C01812=1233.003,73.028,-45.498,-178.669,5.411,148.541
C01813=1233.007,72.779,-45.481,-178.672,5.410,148.542
C01814=1233.012,72.530,-45.463,-178.674,5.409,148.542
C01815=1233.017,72.280,-45.445,-178.677,5.409,148.543
C01816=1233.022,72.031,-45.427,-178.679,5.408,148.544
C01817=1233.027,71.782,-45.409,-178.682,5.408,148.544
C01818=1233.031,71.532,-45.393,-178.684,5.407,148.545
C01819=1233.036,71.283,-45.375,-178.687,5.406,148.545
C01820=1233.041,71.033,-45.358,-178.689,5.406,148.546
C01821=1233.047,70.785,-45.340,-178.692,5.405,148.547
C01822=1233.051,70.536,-45.323,-178.695,5.404,148.547
C01823=1233.056,70.286,-45.305,-178.697,5.404,148.548
C01824=1233.061,70.037,-45.287,-178.700,5.403,148.549
C01825=1233.066,69.787,-45.270,-178.702,5.402,148.549
C01826=1233.070,69.538,-45.253,-178.705,5.402,148.550
C01827=1233.076,69.289,-45.235,-178.707,5.401,148.550
C01828=1233.081,69.039,-45.217,-178.710,5.400,148.551
C01829=1233.085,68.790,-45.201,-178.712,5.400,148.552
C01830=1233.090,68.541,-45.183,-178.715,5.399,148.552
C01831=1233.095,68.291,-45.165,-178.718,5.399,148.553
C01832=1233.100,68.042,-45.147,-178.720,5.398,148.553
C01833=1233.105,67.792,-45.131,-178.722,5.397,148.554
C01834=1233.109,67.543,-45.113,-178.725,5.397,148.555
C01835=1233.115,67.293,-45.096,-178.728,5.396,148.555
C01836=1233.119,67.044,-45.078,-178.730,5.396,148.556
C01837=1233.124,66.795,-45.061,-178.732,5.396,148.557
C01838=1233.130,66.546,-45.043,-178.735,5.395,148.557
C01839=1233.134,66.297,-45.027,-178.737,5.394,148.558
C01840=1233.139,66.048,-45.009,-178.740,5.394,148.558
C01841=1233.143,65.798,-44.992,-178.742,5.393,148.559
C01842=1233.149,65.548,-44.975,-178.745,5.392,148.560
C01843=1233.154,65.299,-44.957,-178.748,5.392,148.560
C01844=1233.158,65.050,-44.940,-178.750,5.391,148.561
C01845=1233.163,64.800,-44.922,-178.752,5.390,148.562
C01846=1233.168,64.551,-44.905,-178.755,5.390,148.562
C01847=1233.173,64.302,-44.889,-178.758,5.389,148.563
C01848=1233.178,64.053,-44.871,-178.760,5.388,148.564
C01849=1233.183,63.803,-44.854,-178.763,5.388,148.564
C01850=1233.188,63.553,-44.837,-178.766,5.387,148.565
C01851=1233.193,63.304,-44.819,-178.768,5.387,148.566
C01852=1233.197,63.055,-44.802,-178.770,5.386,148.566
C01853=1233.203,62.805,-44.785,-178.773,5.385,148.567
C01854=1233.207,62.557,-44.768,-178.776,5.385,148.567
C01855=1233.213,62.307,-44.750,-178.778,5.384,148.568
C01856=1233.217,62.058,-44.734,-178.781,5.383,148.569
C01857=1233.222,61.808,-44.716,-178.784,5.383,148.569
C01858=1233.227,61.559,-44.699,-178.786,5.382,148.570
C01859=1233.232,61.309,-44.682,-178.788,5.382,148.571
C01860=1233.237,61.060,-44.665,-178.790,5.382,148.571
C01861=1233.242,60.811,-44.648,-178.793,5.381,148.572
C01862=1233.247,60.561,-44.630,-178.796,5.380,148.572
C01863=1233.251,60.312,-44.614,-178.798,5.380,148.573
C01864=1233.257,60.062,-44.596,-178.801,5.379,148.574
C01865=1233.262,59.813,-44.580,-178.804,5.379,148.574
C01866=1233.267,59.564,-44.562,-178.806,5.378,148.575
C01867=1233.271,59.315,-44.545,-178.809,5.377,148.576
C01868=1233.276,59.065,-44.528,-178.811,5.377,148.576
C01869=1233.281,58.815,-44.511,-178.814,5.376,148.577
C01870=1233.287,58.566,-44.495,-178.816,5.375,148.578
C01871=1233.291,58.317,-44.477,-178.819,5.375,148.578
C01872=1233.296,58.068,-44.460,-178.821,5.374,148.579
C01873=1233.300,57.818,-44.443,-178.824,5.374,148.580
C01874=1233.305,57.569,-44.427,-178.826,5.374,148.580
C01875=1233.311,57.319,-44.410,-178.829,5.373,148.581
C01876=1233.315,57.070,-44.393,-178.831,5.373,148.582
C01877=1233.320,56.820,-44.376,-178.834,5.372,148.582
C01878=1233.325,56.571,-44.359,-178.836,5.371,148.583
C01879=1233.330,56.322,-44.341,-178.839,5.371,148.583
C01880=1233.335,56.053,-44.324,-178.842,5.370,148.584
C01881=1233.341,55.785,-44.306,-178.844,5.369,148.585
C01882=1233.346,55.516,-44.288,-178.847,5.369,148.586
C01883=1233.351,55.248,-44.270,-178.850,5.369,148.586
C01884=1233.356,54.999,-44.253,-178.853,5.368,148.587
C01885=1233.361,54.749,-44.236,-178.855,5.367,148.587
C01886=1233.366,54.499,-44.219,-178.857,5.367,148.588
C01887=1233.371,54.251,-44.202,-178.860,5.366,148.589
C01888=1233.376,54.001,-44.186,-178.863,5.365,148.589
C01889=1233.381,53.751,-44.168,-178.865,5.365,148.590
C01890=1233.385,53.502,-44.152,-178.868,5.364,148.591
C01891=1233.390,53.253,-44.136,-178.870,5.364,148.591
C01892=1233.396,53.003,-44.118,-178.873,5.364,148.592
C01893=1233.400,52.754,-44.102,-178.875,5.363,148.593
C01894=1233.405,52.505,-44.085,-178.878,5.363,148.593
C01895=1233.410,52.255,-44.068,-178.880,5.362,148.594
C01896=1233.415,52.006,-44.051,-178.883,5.361,148.594
C01897=1233.420,51.757,-44.035,-178.885,5.361,148.595
C01898=1233.425,51.507,-44.018,-178.888,5.360,148.596
C01899=1233.430,51.258,-44.001,-178.891,5.359,148.596
C01900=1233.435,51.009,-43.985,-178.893,5.359,148.597
C01901=1233.440,50.759,-43.968,-178.896,5.358,148.598
C01902=1233.445,50.510,-43.951,-178.898,5.359,148.598
C01903=1233.450,50.261,-43.935,-178.900,5.358,148.599
C01904=1233.454,50.011,-43.918,-178.903,5.357,148.600
C01905=1233.459,49.762,-43.901,-178.905,5.357,148.600
C01906=1233.465,49.512,-43.885,-178.908,5.356,148.601
C01907=1233.469,49.263,-43.868,-178.911,5.355,148.602
C01908=1233.474,49.013,-43.852,-178.913,5.355,148.602
C01909=1233.479,48.764,-43.835,-178.916,5.354,148.603
C01910=1233.484,48.515,-43.818,-178.918,5.354,148.604
C01911=1233.488,48.265,-43.801,-178.921,5.354,148.604
C01912=1233.493,48.016,-43.785,-178.923,5.353,148.605
C01913=1233.499,47.766,-43.769,-178.926,5.353,148.606
C01914=1233.504,47.517,-43.752,-178.928,5.352,148.606
C01915=1233.509,47.268,-43.736,-178.931,5.352,148.607
C01916=1233.513,47.018,-43.719,-178.934,5.351,148.608
C01917=1233.518,46.769,-43.703,-178.936,5.350,148.608
C01918=1233.524,46.519,-43.686,-178.938,5.350,148.609
C01919=1233.528,46.269,-43.669,-178.941,5.350,148.609
C01920=1233.533,46.021,-43.653,-178.943,5.349,148.610
C01921=1233.538,45.771,-43.636,-178.946,5.349,148.611
C01922=1233.543,45.522,-43.621,-178.948,5.348,148.611
C01923=1233.548,45.272,-43.604,-178.951,5.347,148.612
C01924=1233.553,45.023,-43.587,-178.954,5.347,148.613
C01925=1233.558,44.773,-43.571,-178.956,5.346,148.613
C01926=1233.563,44.524,-43.555,-178.959,5.346,148.614
C01927=1233.568,44.275,-43.538,-178.961,5.346,148.615
C01928=1233.572,44.025,-43.522,-178.964,5.345,148.615
C01929=1233.578,43.776,-43.506,-178.966,5.345,148.616
C01930=1233.583,43.526,-43.489,-178.969,5.344,148.617
C01931=1233.588,43.277,-43.473,-178.971,5.343,148.617
C01932=1233.593,43.027,-43.457,-178.974,5.343,148.618
C01933=1233.597,42.778,-43.440,-178.976,5.342,148.619
C01934=1233.602,42.529,-43.424,-178.979,5.342,148.619
C01935=1233.607,42.279,-43.408,-178.981,5.342,148.620
C01936=1233.612,42.030,-43.391,-178.984,5.341,148.621
C01937=1233.617,41.780,-43.375,-178.986,5.341,148.621
C01938=1233.622,41.531,-43.359,-178.989,5.340,148.622
C01939=1233.626,41.282,-43.342,-178.992,5.340,148.623
C01940=1233.633,41.032,-43.326,-178.994,5.339,148.623
C01941=1233.637,40.783,-43.310,-178.996,5.339,148.624
C01942=1233.642,40.533,-43.294,-178.999,5.339,148.625
C01943=1233.647,40.284,-43.277,-179.002,5.338,148.625
C01944=1233.652,40.035,-43.261,-179.004,5.338,148.626
C01945=1233.657,39.785,-43.245,-179.007,5.337,148.627
C01946=1233.662,39.536,-43.229,-179.010,5.337,148.627
C01947=1233.667,39.286,-43.213,-179.012,5.336,148.628
C01948=1233.672,39.037,-43.197,-179.014,5.336,148.628
C01949=1233.677,38.787,-43.181,-179.016,5.335,148.629
C01950=1233.682,38.538,-43.164,-179.019,5.335,148.630
C01951=1233.686,38.288,-43.148,-179.022,5.334,148.631
C01952=1233.691,38.039,-43.132,-179.024,5.334,148.631
C01953=1233.696,37.789,-43.116,-179.027,5.333,148.632
C01954=1233.701,37.540,-43.100,-179.029,5.333,148.633
C01955=1233.706,37.290,-43.084,-179.032,5.333,148.633
C01956=1233.711,37.042,-43.068,-179.034,5.332,148.634
C01957=1233.716,36.791,-43.052,-179.037,5.332,148.635
C01958=1233.721,36.543,-43.035,-179.040,5.331,148.635
C01959=1233.726,36.293,-43.020,-179.042,5.330,148.636
C01960=1233.731,36.043,-43.004,-179.044,5.331,148.637
C01961=1233.736,35.794,-42.987,-179.047,5.330,148.637
C01962=1233.741,35.544,-42.971,-179.050,5.330,148.638
C01963=1233.746,35.296,-42.955,-179.052,5.329,148.639
C01964=1233.751,35.045,-42.939,-179.055,5.328,148.639
C01965=1233.756,34.796,-42.924,-179.058,5.328,148.640
C01966=1233.760,34.547,-42.908,-179.060,5.328,148.641
C01967=1233.766,34.297,-42.892,-179.062,5.328,148.641
C01968=1233.771,34.049,-42.876,-179.065,5.327,148.642
C01969=1233.775,33.799,-42.860,-179.067,5.326,148.642
C01970=1233.781,33.549,-42.844,-179.070,5.326,148.643
C01971=1233.785,33.300,-42.827,-179.072,5.325,148.644
C01972=1233.791,33.050,-42.812,-179.074,5.325,148.644
C01973=1233.796,32.801,-42.796,-179.077,5.325,148.645
C01974=1233.800,32.551,-42.780,-179.080,5.324,148.646
C01975=1233.805,32.302,-42.765,-179.082,5.324,148.647
C01976=1233.810,32.052,-42.749,-179.085,5.323,148.647
C01977=1233.815,31.803,-42.732,-179.087,5.323,148.648
C01978=1233.820,31.554,-42.717,-179.090,5.323,148.649
C01979=1233.825,31.304,-42.701,-179.092,5.322,148.649
C01980=1233.831,31.054,-42.685,-179.095,5.322,148.650
C01981=1233.835,30.805,-42.669,-179.098,5.321,148.651
C01982=1233.840,30.556,-42.654,-179.100,5.320,148.651
C01983=1233.845,30.307,-42.638,-179.102,5.321,148.652
C01984=1233.850,30.037,-42.621,-179.105,5.320,148.653
C01985=1233.856,29.769,-42.604,-179.108,5.320,148.653
C01986=1233.861,29.500,-42.587,-179.111,5.319,148.654
C01987=1233.867,29.232,-42.570,-179.113,5.319,148.655
C01988=1233.871,28.983,-42.555,-179.116,5.318,148.656
C01989=1233.876,28.733,-42.539,-179.119,5.318,148.656
C01990=1233.881,28.484,-42.522,-179.121,5.317,148.657
C01991=1233.887,28.235,-42.507,-179.123,5.317,148.658
C01992=1233.891,27.984,-42.491,-179.126,5.317,148.658
C01993=1233.896,27.735,-42.476,-179.129,5.316,148.659
C01994=1233.901,27.486,-42.460,-179.131,5.316,148.660
C01995=1233.906,27.236,-42.444,-179.134,5.315,148.660
C01996=1233.911,26.987,-42.428,-179.136,5.315,148.661
C01997=1233.916,26.738,-42.413,-179.139,5.315,148.662
C01998=1233.921,26.488,-42.397,-179.141,5.314,148.662
C01999=1233.926,26.238,-42.381,-179.144,5.314,148.663
C02000=1233.932,25.989,-42.366,-179.146,5.314,148.664
C02001=1233.936,25.739,-42.350,-179.148,5.313,148.664
C02002=1233.941,25.490,-42.335,-179.151,5.313,148.665
C02003=1233.946,25.240,-42.319,-179.154,5.312,148.666
C02004=1233.951,24.991,-42.304,-179.156,5.312,148.666
C02005=1233.955,24.742,-42.288,-179.158,5.312,148.667
C02006=1233.961,24.492,-42.272,-179.161,5.311,148.668
C02007=1233.966,24.243,-42.256,-179.164,5.311,148.668
C02008=1233.970,23.993,-42.241,-179.166,5.310,148.669
C02009=1233.976,23.744,-42.225,-179.169,5.310,148.670
C02010=1233.981,23.494,-42.210,-179.171,5.310,148.670
C02011=1233.986,23.245,-42.195,-179.174,5.309,148.671
C02012=1233.990,22.995,-42.179,-179.176,5.309,148.672
C02013=1233.996,22.746,-42.163,-179.179,5.308,148.672
C02014=1234.001,22.497,-42.148,-179.181,5.308,148.673
C02015=1234.006,22.247,-42.133,-179.184,5.308,148.674
C02016=1234.010,21.998,-42.117,-179.186,5.307,148.674
C02017=1234.015,21.748,-42.102,-179.189,5.307,148.675
C02018=1234.021,21.499,-42.086,-179.192,5.306,148.676
C02019=1234.025,21.250,-42.071,-179.194,5.306,148.676
C02020=1234.030,21.000,-42.055,-179.196,5.306,148.677
C02021=1234.036,20.750,-42.040,-179.199,5.305,148.678
C02022=1234.040,20.501,-42.025,-179.202,5.305,148.678
C02023=1234.046,20.251,-42.010,-179.204,5.305,148.679
C02024=1234.050,20.001,-41.994,-179.206,5.305,148.680
C02025=1234.055,19.752,-41.979,-179.209,5.304,148.681
C02026=1234.061,19.502,-41.963,-179.212,5.303,148.681
C02027=1234.065,19.253,-41.948,-179.214,5.303,148.682
C02028=1234.071,19.004,-41.933,-179.216,5.303,148.683
C02029=1234.075,18.754,-41.917,-179.219,5.303,148.683
C02030=1234.080,18.505,-41.902,-179.222,5.302,148.684
C02031=1234.085,18.256,-41.887,-179.224,5.302,148.685
C02032=1234.091,18.006,-41.872,-179.226,5.302,148.685
C02033=1234.095,17.757,-41.857,-179.229,5.301,148.686
C02034=1234.101,17.507,-41.841,-179.232,5.301,148.687
C02035=1234.105,17.257,-41.825,-179.234,5.300,148.687
C02036=1234.110,17.008,-41.810,-179.236,5.300,148.688
C02037=1234.115,16.759,-41.795,-179.239,5.300,148.689
C02038=1234.120,16.509,-41.781,-179.242,5.299,148.689
C02039=1234.126,16.259,-41.765,-179.244,5.299,148.690
C02040=1234.130,16.010,-41.750,-179.246,5.299,148.691
C02041=1234.135,15.760,-41.734,-179.249,5.299,148.691
C02042=1234.140,15.511,-41.719,-179.252,5.298,148.692
C02043=1234.146,15.261,-41.704,-179.254,5.297,148.693
C02044=1234.150,15.012,-41.689,-179.256,5.298,148.694
C02045=1234.156,14.763,-41.674,-179.259,5.297,148.694
C02046=1234.160,14.514,-41.659,-179.262,5.297,148.695
C02047=1234.166,14.264,-41.644,-179.264,5.296,148.696
C02048=1234.170,14.014,-41.628,-179.266,5.296,148.696
C02049=1234.175,13.765,-41.613,-179.269,5.296,148.697
C02050=1234.180,13.515,-41.598,-179.272,5.295,148.698
C02051=1234.185,13.266,-41.583,-179.274,5.295,148.698
C02052=1234.190,13.016,-41.568,-179.276,5.295,148.699
C02053=1234.195,12.767,-41.553,-179.279,5.294,148.700
C02054=1234.201,12.517,-41.538,-179.282,5.294,148.700
C02055=1234.205,12.268,-41.523,-179.284,5.293,148.701
C02056=1234.210,12.018,-41.507,-179.286,5.294,148.702
C02057=1234.215,11.768,-41.493,-179.289,5.293,148.702
C02058=1234.220,11.519,-41.478,-179.292,5.293,148.703
C02059=1234.225,11.270,-41.462,-179.294,5.292,148.704
C02060=1234.230,11.020,-41.448,-179.296,5.292,148.704
C02061=1234.235,10.771,-41.432,-179.300,5.292,148.705
C02062=1234.240,10.521,-41.417,-179.302,5.292,148.706
C02063=1234.245,10.272,-41.403,-179.305,5.291,148.707
C02064=1234.250,10.022,-41.387,-179.307,5.291,148.707
C02065=1234.255,9.773,-41.373,-179.310,5.291,148.708
C02066=1234.260,9.524,-41.358,-179.312,5.290,148.709
C02067=1234.265,9.274,-41.343,-179.314,5.290,148.710
C02068=1234.270,9.024,-41.328,-179.317,5.290,148.710
C02069=1234.274,8.775,-41.313,-179.320,5.289,148.711
C02070=1234.280,8.525,-41.298,-179.322,5.289,148.712
C02071=1234.285,8.275,-41.283,-179.324,5.289,148.712
C02072=1234.290,8.026,-41.269,-179.327,5.289,148.713
C02073=1234.295,7.776,-41.253,-179.330,5.288,148.714
C02074=1234.300,7.527,-41.239,-179.332,5.288,148.714
C02075=1234.305,7.278,-41.224,-179.334,5.288,148.715
C02076=1234.310,7.028,-41.209,-179.337,5.287,148.716
C02077=1234.315,6.778,-41.194,-179.340,5.287,148.716
C02078=1234.320,6.529,-41.180,-179.342,5.287,148.717
C02079=1234.325,6.279,-41.164,-179.344,5.286,148.718
C02080=1234.330,6.030,-41.150,-179.347,5.286,148.718
C02081=1234.335,5.781,-41.135,-179.350,5.285,148.719
C02082=1234.340,5.531,-41.121,-179.352,5.286,148.720
C02083=1234.345,5.281,-41.105,-179.354,5.285,148.720
C02084=1234.350,5.032,-41.091,-179.357,5.285,148.721
C02085=1234.355,4.783,-41.076,-179.359,5.285,148.722
C02086=1234.360,4.533,-41.062,-179.362,5.284,148.723
C02087=1234.365,4.284,-41.046,-179.364,5.284,148.723
C02088=1234.370,4.015,-41.030,-179.367,5.283,148.724
C02089=1234.376,3.746,-41.015,-179.370,5.283,148.725
C02090=1234.381,3.477,-40.998,-179.372,5.283,148.726
C02091=1234.387,3.207,-40.983,-179.375,5.283,148.726
C02092=1234.391,2.958,-40.968,-179.378,5.282,148.727
C02093=1234.396,2.709,-40.954,-179.380,5.282,148.728
C02094=1234.402,2.459,-40.938,-179.382,5.282,148.728
C02095=1234.407,2.210,-40.924,-179.385,5.282,148.729
C02096=1234.412,1.961,-40.910,-179.388,5.281,148.730
C02097=1234.417,1.711,-40.895,-179.390,5.281,148.730
C02098=1234.422,1.462,-40.881,-179.392,5.281,148.731
C02099=1234.428,1.212,-40.866,-179.395,5.280,148.732
C02100=1234.432,0.963,-40.851,-179.398,5.280,148.732
C02101=1234.437,0.713,-40.837,-179.400,5.280,148.733
C02102=1234.442,0.463,-40.823,-179.403,5.280,148.734
C02103=1234.447,0.214,-40.808,-179.406,5.279,148.735
C02104=1234.452,-0.036,-40.793,-179.408,5.280,148.735
C02105=1234.457,-0.286,-40.778,-179.410,5.279,148.736
C02106=1234.462,-0.535,-40.764,-179.413,5.278,148.737
C02107=1234.467,-0.784,-40.749,-179.415,5.279,148.737
C02108=1234.472,-1.034,-40.735,-179.418,5.278,148.738
C02109=1234.477,-1.284,-40.721,-179.420,5.278,148.739
C02110=1234.482,-1.532,-40.706,-179.423,5.277,148.740
C02111=1234.487,-1.782,-40.692,-179.425,5.277,148.740
C02112=1234.492,-2.032,-40.677,-179.428,5.277,148.741
C02113=1234.498,-2.282,-40.663,-179.430,5.276,148.742
C02114=1234.503,-2.531,-40.648,-179.433,5.277,148.742
C02115=1234.507,-2.781,-40.633,-179.435,5.276,148.743
C02116=1234.512,-3.030,-40.619,-179.438,5.276,148.744
C02117=1234.517,-3.280,-40.605,-179.440,5.276,148.744
C02118=1234.522,-3.530,-40.590,-179.443,5.275,148.745
C02119=1234.528,-3.779,-40.576,-179.445,5.275,148.746
C02120=1234.533,-4.028,-40.562,-179.447,5.275,148.746
C02121=1234.537,-4.277,-40.547,-179.450,5.275,148.747
C02122=1234.542,-4.527,-40.533,-179.453,5.274,148.748
C02123=1234.547,-4.777,-40.519,-179.455,5.274,148.749
C02124=1234.552,-5.027,-40.504,-179.457,5.274,148.749
C02125=1234.557,-5.276,-40.490,-179.460,5.273,148.750
C02126=1234.562,-5.526,-40.476,-179.462,5.274,148.751
C02127=1234.567,-5.774,-40.461,-179.465,5.273,148.752
C02128=1234.573,-6.024,-40.446,-179.468,5.273,148.752
C02129=1234.578,-6.274,-40.432,-179.471,5.272,148.753
C02130=1234.583,-6.524,-40.418,-179.473,5.273,148.754
C02131=1234.588,-6.774,-40.404,-179.475,5.272,148.754
C02132=1234.593,-7.023,-40.389,-179.478,5.272,148.755
C02133=1234.599,-7.272,-40.375,-179.480,5.272,148.756
C02134=1234.604,-7.522,-40.361,-179.483,5.271,148.756
C02135=1234.608,-7.771,-40.347,-179.485,5.271,148.757
C02136=1234.613,-8.021,-40.333,-179.487,5.271,148.758
C02137=1234.618,-8.271,-40.319,-179.490,5.271,148.758
C02138=1234.623,-8.521,-40.305,-179.493,5.270,148.759
C02139=1234.628,-8.770,-40.291,-179.495,5.270,148.760
C02140=1234.633,-9.019,-40.276,-179.497,5.270,148.761
C02141=1234.638,-9.269,-40.262,-179.500,5.269,148.761
C02142=1234.643,-9.519,-40.248,-179.502,5.270,148.762
C02143=1234.648,-9.768,-40.234,-179.505,5.269,148.763
C02144=1234.654,-10.017,-40.220,-179.507,5.269,148.763
C02145=1234.658,-10.267,-40.205,-179.510,5.269,148.764
C02146=1234.663,-10.517,-40.191,-179.512,5.268,148.765
C02147=1234.668,-10.767,-40.177,-179.515,5.268,148.765
C02148=1234.674,-11.016,-40.163,-179.517,5.268,148.766
C02149=1234.679,-11.265,-40.149,-179.520,5.268,148.767
C02150=1234.684,-11.515,-40.134,-179.523,5.267,148.768
C02151=1234.689,-11.765,-40.120,-179.525,5.268,148.768
C02152=1234.694,-12.013,-40.107,-179.528,5.267,148.769
C02153=1234.699,-12.263,-40.092,-179.530,5.267,148.770
C02154=1234.704,-12.513,-40.078,-179.532,5.267,148.770
C02155=1234.708,-12.762,-40.064,-179.535,5.266,148.771
C02156=1234.714,-13.011,-40.050,-179.537,5.267,148.772
C02157=1234.719,-13.261,-40.036,-179.540,5.266,148.773
C02158=1234.724,-13.511,-40.021,-179.542,5.266,148.773
C02159=1234.729,-13.761,-40.008,-179.544,5.266,148.774
C02160=1234.734,-14.010,-39.995,-179.547,5.265,148.775
C02161=1234.739,-14.260,-39.980,-179.550,5.265,148.775
C02162=1234.744,-14.509,-39.966,-179.552,5.265,148.776
C02163=1234.749,-14.759,-39.952,-179.554,5.265,148.777
C02164=1234.754,-15.008,-39.938,-179.557,5.264,148.777
C02165=1234.759,-15.258,-39.924,-179.559,5.264,148.778
C02166=1234.764,-15.508,-39.911,-179.562,5.264,148.779
C02167=1234.769,-15.757,-39.897,-179.565,5.264,148.780
C02168=1234.774,-16.007,-39.882,-179.567,5.264,148.780
C02169=1234.779,-16.256,-39.868,-179.570,5.264,148.781
C02170=1234.784,-16.506,-39.854,-179.572,5.263,148.782
C02171=1234.789,-16.755,-39.841,-179.574,5.263,148.782
C02172=1234.794,-17.005,-39.827,-179.577,5.263,148.783
C02173=1234.799,-17.255,-39.813,-179.580,5.262,148.784
C02174=1234.805,-17.504,-39.799,-179.582,5.263,148.785
C02175=1234.810,-17.754,-39.785,-179.585,5.262,148.785
C02176=1234.814,-18.003,-39.771,-179.587,5.262,148.786
C02177=1234.820,-18.252,-39.758,-179.589,5.262,148.787
C02178=1234.825,-18.502,-39.743,-179.592,5.261,148.787
C02179=1234.830,-18.752,-39.730,-179.594,5.262,148.788
C02180=1234.835,-19.001,-39.716,-179.597,5.261,148.789
C02181=1234.840,-19.251,-39.702,-179.599,5.261,148.789
C02182=1234.845,-19.501,-39.688,-179.601,5.261,148.790
C02183=1234.851,-19.750,-39.675,-179.604,5.260,148.791
C02184=1234.855,-20.000,-39.661,-179.607,5.260,148.791
C02185=1234.860,-20.249,-39.647,-179.609,5.261,148.792
C02186=1234.866,-20.499,-39.634,-179.612,5.260,148.793
C02187=1234.870,-20.748,-39.620,-179.614,5.260,148.794
C02188=1234.876,-20.997,-39.606,-179.617,5.260,148.795
C02189=1234.881,-21.248,-39.592,-179.619,5.259,148.795
C02190=1234.886,-21.497,-39.578,-179.621,5.260,148.796
C02191=1234.891,-21.746,-39.565,-179.624,5.259,148.797
C02192=1234.896,-22.016,-39.550,-179.627,5.259,148.797
C02193=1234.902,-22.286,-39.536,-179.629,5.259,148.798
C02194=1234.907,-22.555,-39.521,-179.632,5.259,148.799
C02195=1234.913,-22.824,-39.506,-179.635,5.258,148.800
C02196=1234.917,-23.073,-39.492,-179.637,5.258,148.800
C02197=1234.923,-23.323,-39.479,-179.639,5.258,148.801
C02198=1234.928,-23.572,-39.465,-179.642,5.257,148.802
C02199=1234.933,-23.822,-39.451,-179.644,5.258,148.802
C02200=1234.938,-24.071,-39.438,-179.647,5.257,148.803
C02201=1234.943,-24.321,-39.424,-179.649,5.257,148.804
C02202=1234.948,-24.571,-39.411,-179.652,5.257,148.805
C02203=1234.953,-24.820,-39.397,-179.655,5.257,148.805
C02204=1234.958,-25.070,-39.384,-179.657,5.256,148.806
C02205=1234.963,-25.319,-39.370,-179.659,5.257,148.807
C02206=1234.968,-25.569,-39.357,-179.662,5.256,148.808
C02207=1234.974,-25.818,-39.343,-179.664,5.257,148.808
C02208=1234.979,-26.069,-39.329,-179.667,5.256,148.809
C02209=1234.983,-26.318,-39.316,-179.669,5.255,148.810
C02210=1234.989,-26.568,-39.303,-179.672,5.256,148.810
C02211=1234.993,-26.817,-39.289,-179.674,5.255,148.811
C02212=1234.999,-27.067,-39.276,-179.677,5.255,148.812
C02213=1235.004,-27.316,-39.261,-179.679,5.255,148.812
C02214=1235.009,-27.566,-39.249,-179.682,5.255,148.813
C02215=1235.014,-27.815,-39.234,-179.684,5.255,148.814
C02216=1235.019,-28.065,-39.222,-179.686,5.254,148.814
C02217=1235.024,-28.314,-39.208,-179.690,5.254,148.815
C02218=1235.029,-28.564,-39.195,-179.692,5.255,148.816
C02219=1235.034,-28.813,-39.181,-179.694,5.254,148.817
C02220=1235.039,-29.063,-39.168,-179.696,5.254,148.818
C02221=1235.045,-29.313,-39.155,-179.699,5.254,148.818
C02222=1235.049,-29.562,-39.141,-179.702,5.253,148.819
C02223=1235.055,-29.812,-39.128,-179.704,5.254,148.820
C02224=1235.059,-30.062,-39.114,-179.706,5.253,148.820
C02225=1235.065,-30.311,-39.101,-179.709,5.253,148.821
C02226=1235.069,-30.561,-39.088,-179.711,5.253,148.822
C02227=1235.075,-30.810,-39.074,-179.714,5.252,148.822
C02228=1235.079,-31.060,-39.061,-179.716,5.253,148.823
C02229=1235.085,-31.310,-39.048,-179.719,5.252,148.824
C02230=1235.089,-31.559,-39.034,-179.721,5.253,148.824
C02231=1235.095,-31.809,-39.021,-179.723,5.252,148.825
C02232=1235.100,-32.058,-39.008,-179.726,5.251,148.826
C02233=1235.105,-32.308,-38.994,-179.729,5.252,148.827
C02234=1235.110,-32.557,-38.981,-179.731,5.252,148.828
C02235=1235.116,-32.808,-38.968,-179.733,5.252,148.828
C02236=1235.121,-33.056,-38.955,-179.736,5.251,148.829
C02237=1235.126,-33.307,-38.941,-179.739,5.251,148.830
C02238=1235.131,-33.556,-38.928,-179.741,5.251,148.830
C02239=1235.135,-33.805,-38.915,-179.743,5.251,148.831
C02240=1235.141,-34.055,-38.901,-179.745,5.251,148.832
C02241=1235.146,-34.305,-38.889,-179.748,5.251,148.832
C02242=1235.151,-34.555,-38.875,-179.751,5.250,148.833
C02243=1235.156,-34.804,-38.862,-179.753,5.250,148.834
C02244=1235.161,-35.054,-38.848,-179.756,5.250,148.835
C02245=1235.167,-35.303,-38.836,-179.758,5.250,148.835
C02246=1235.171,-35.553,-38.823,-179.760,5.250,148.836
C02247=1235.177,-35.802,-38.809,-179.763,5.249,148.837
C02248=1235.181,-36.052,-38.796,-179.766,5.250,148.838
C02249=1235.187,-36.302,-38.783,-179.768,5.249,148.838
C02250=1235.192,-36.551,-38.770,-179.770,5.250,148.839
C02251=1235.197,-36.801,-38.757,-179.773,5.249,148.840
C02252=1235.202,-37.050,-38.743,-179.776,5.249,148.840
C02253=1235.207,-37.300,-38.730,-179.778,5.249,148.841
C02254=1235.212,-37.549,-38.718,-179.780,5.248,148.842
C02255=1235.218,-37.799,-38.705,-179.782,5.249,148.842
C02256=1235.222,-38.049,-38.692,-179.785,5.248,148.843
C02257=1235.227,-38.298,-38.679,-179.787,5.249,148.844
C02258=1235.232,-38.548,-38.665,-179.790,5.248,148.845
C02259=1235.237,-38.797,-38.652,-179.793,5.248,148.845
C02260=1235.243,-39.047,-38.640,-179.795,5.248,148.846
C02261=1235.248,-39.297,-38.626,-179.797,5.247,148.847
C02262=1235.253,-39.546,-38.613,-179.799,5.248,148.847
C02263=1235.258,-39.796,-38.600,-179.802,5.248,148.848
C02264=1235.263,-40.046,-38.587,-179.805,5.247,148.849
C02265=1235.268,-40.295,-38.575,-179.807,5.247,148.850
C02266=1235.273,-40.545,-38.562,-179.810,5.247,148.850
C02267=1235.279,-40.795,-38.548,-179.812,5.247,148.851
C02268=1235.284,-41.043,-38.535,-179.815,5.247,148.852
C02269=1235.288,-41.294,-38.522,-179.817,5.247,148.852
C02270=1235.293,-41.543,-38.510,-179.819,5.247,148.853
C02271=1235.299,-41.792,-38.496,-179.822,5.246,148.854
C02272=1235.304,-42.042,-38.483,-179.824,5.246,148.855
C02273=1235.309,-42.292,-38.471,-179.827,5.246,148.855
C02274=1235.314,-42.541,-38.458,-179.829,5.246,148.856
C02275=1235.319,-42.791,-38.445,-179.832,5.246,148.857
C02276=1235.324,-43.041,-38.432,-179.834,5.246,148.857
C02277=1235.329,-43.290,-38.419,-179.836,5.246,148.858
C02278=1235.334,-43.540,-38.406,-179.839,5.245,148.859
C02279=1235.340,-43.790,-38.393,-179.842,5.246,148.860
C02280=1235.345,-44.039,-38.381,-179.844,5.245,148.860
C02281=1235.350,-44.289,-38.368,-179.846,5.246,148.861
C02282=1235.355,-44.538,-38.355,-179.849,5.245,148.862
C02283=1235.360,-44.788,-38.342,-179.851,5.245,148.863
C02284=1235.365,-45.038,-38.329,-179.854,5.245,148.863
C02285=1235.370,-45.287,-38.316,-179.856,5.244,148.864
C02286=1235.375,-45.537,-38.304,-179.858,5.245,148.865
C02287=1235.381,-45.787,-38.292,-179.861,5.244,148.865
C02288=1235.385,-46.037,-38.279,-179.863,5.244,148.866
C02289=1235.391,-46.286,-38.266,-179.866,5.244,148.867
C02290=1235.396,-46.536,-38.253,-179.868,5.244,148.867
C02291=1235.401,-46.786,-38.240,-179.871,5.244,148.868
C02292=1235.406,-47.035,-38.228,-179.873,5.244,148.869
C02293=1235.411,-47.284,-38.215,-179.876,5.244,148.870
C02294=1235.416,-47.534,-38.202,-179.879,5.244,148.870
C02295=1235.421,-47.784,-38.189,-179.881,5.244,148.871
C02296=1235.427,-48.053,-38.175,-179.883,5.243,148.872
C02297=1235.432,-48.323,-38.162,-179.886,5.243,148.873
C02298=1235.438,-48.593,-38.148,-179.889,5.244,148.874
C02299=1235.444,-48.862,-38.135,-179.891,5.243,148.874
C02300=1235.448,-49.112,-38.122,-179.893,5.243,148.875
C02301=1235.453,-49.362,-38.109,-179.896,5.243,148.876
C02302=1235.458,-49.611,-38.097,-179.899,5.242,148.876
C02303=1235.464,-49.861,-38.085,-179.901,5.243,148.877
C02304=1235.469,-50.111,-38.071,-179.903,5.242,148.878
C02305=1235.474,-50.361,-38.059,-179.905,5.243,148.878
C02306=1235.479,-50.610,-38.046,-179.908,5.242,148.879
C02307=1235.484,-50.859,-38.033,-179.910,5.242,148.880
C02308=1235.490,-51.109,-38.022,-179.913,5.242,148.881
C02309=1235.494,-51.359,-38.009,-179.915,5.243,148.881
C02310=1235.500,-51.608,-37.996,-179.918,5.242,148.882
C02311=1235.505,-51.858,-37.983,-179.921,5.242,148.883
C02312=1235.510,-52.108,-37.972,-179.923,5.242,148.884
C02313=1235.515,-52.358,-37.959,-179.926,5.241,148.884
C02314=1235.520,-52.607,-37.946,-179.928,5.242,148.885
C02315=1235.525,-52.856,-37.933,-179.930,5.241,148.886
C02316=1235.530,-53.106,-37.921,-179.932,5.242,148.886
C02317=1235.535,-53.356,-37.909,-179.935,5.241,148.887
C02318=1235.541,-53.605,-37.896,-179.937,5.241,148.888
C02319=1235.545,-53.856,-37.884,-179.940,5.241,148.889
C02320=1235.550,-54.105,-37.871,-179.942,5.241,148.889
C02321=1235.556,-54.354,-37.859,-179.945,5.241,148.890
C02322=1235.561,-54.604,-37.846,-179.947,5.240,148.891
C02323=1235.566,-54.853,-37.834,-179.949,5.241,148.891
C02324=1235.571,-55.103,-37.821,-179.952,5.240,148.892
C02325=1235.576,-55.353,-37.809,-179.955,5.241,148.893
C02326=1235.581,-55.603,-37.797,-179.957,5.240,148.894
C02327=1235.586,-55.852,-37.784,-179.959,5.241,148.894
C02328=1235.592,-56.102,-37.772,-179.962,5.240,148.895
C02329=1235.597,-56.351,-37.760,-179.964,5.241,148.896
C02330=1235.601,-56.601,-37.747,-179.967,5.240,148.896
C02331=1235.607,-56.851,-37.735,-179.969,5.240,148.897
C02332=1235.612,-57.101,-37.722,-179.972,5.240,148.898
C02333=1235.617,-57.350,-37.710,-179.974,5.239,148.899
C02334=1235.623,-57.600,-37.698,-179.976,5.240,148.899
C02335=1235.628,-57.849,-37.685,-179.979,5.239,148.900
C02336=1235.633,-58.099,-37.673,-179.981,5.240,148.901
C02337=1235.638,-58.348,-37.661,-179.984,5.239,148.901
C02338=1235.643,-58.599,-37.649,-179.986,5.239,148.902
C02339=1235.647,-58.848,-37.636,-179.988,5.239,148.903
C02340=1235.653,-59.097,-37.624,-179.991,5.239,148.904
C02341=1235.658,-59.347,-37.612,-179.993,5.239,148.904
C02342=1235.663,-59.597,-37.599,-179.996,5.239,148.905
C02343=1235.669,-59.847,-37.588,-179.998,5.239,148.906
C02344=1235.674,-60.096,-37.575,179.999,5.239,148.907
C02345=1235.679,-60.346,-37.563,179.997,5.239,148.907
C02346=1235.684,-60.595,-37.550,179.995,5.239,148.908
C02347=1235.689,-60.846,-37.538,179.992,5.239,148.909
C02348=1235.693,-61.095,-37.526,179.989,5.238,148.909
C02349=1235.699,-61.345,-37.514,179.987,5.239,148.910
C02350=1235.704,-61.594,-37.502,179.985,5.238,148.911
C02351=1235.709,-61.844,-37.490,179.983,5.238,148.912
C02352=1235.715,-62.093,-37.477,179.980,5.238,148.912
C02353=1235.720,-62.343,-37.465,179.978,5.238,148.913
C02354=1235.725,-62.593,-37.454,179.975,5.238,148.914
C02355=1235.730,-62.842,-37.441,179.973,5.238,148.914
C02356=1235.735,-63.092,-37.430,179.970,5.238,148.915
C02357=1235.740,-63.341,-37.417,179.968,5.238,148.916
C02358=1235.746,-63.591,-37.405,179.966,5.237,148.916
C02359=1235.751,-63.841,-37.392,179.963,5.238,148.917
C02360=1235.756,-64.090,-37.381,179.960,5.238,148.918
C02361=1235.761,-64.340,-37.369,179.958,5.238,148.919
C02362=1235.766,-64.590,-37.357,179.956,5.238,148.920
C02363=1235.772,-64.839,-37.345,179.953,5.238,148.920
C02364=1235.777,-65.089,-37.332,179.951,5.237,148.921
C02365=1235.781,-65.338,-37.321,179.949,5.238,148.922
C02366=1235.786,-65.589,-37.309,179.946,5.237,148.922
C02367=1235.791,-65.838,-37.296,179.943,5.237,148.923
C02368=1235.797,-66.088,-37.284,179.941,5.237,148.924
C02369=1235.801,-66.338,-37.273,179.939,5.237,148.924
C02370=1235.807,-66.587,-37.260,179.937,5.237,148.925
C02371=1235.812,-66.837,-37.248,179.934,5.236,148.926
C02372=1235.817,-67.087,-37.237,179.932,5.237,148.927
C02373=1235.822,-67.336,-37.225,179.929,5.236,148.927
C02374=1235.827,-67.586,-37.213,179.927,5.237,148.928
C02375=1235.833,-67.836,-37.201,179.924,5.236,148.929
C02376=1235.838,-68.085,-37.188,179.922,5.237,148.929
C02377=1235.842,-68.335,-37.177,179.920,5.236,148.930
C02378=1235.849,-68.584,-37.165,179.917,5.236,148.931
C02379=1235.854,-68.834,-37.153,179.915,5.236,148.932
C02380=1235.859,-69.083,-37.141,179.912,5.237,148.932
C02381=1235.864,-69.333,-37.130,179.910,5.236,148.933
C02382=1235.869,-69.583,-37.118,179.907,5.236,148.934
C02383=1235.875,-69.833,-37.106,179.905,5.236,148.935
C02384=1235.879,-70.082,-37.094,179.903,5.236,148.935
C02385=1235.884,-70.332,-37.082,179.900,5.236,148.936
C02386=1235.890,-70.582,-37.070,179.898,5.236,148.937
C02387=1235.895,-70.831,-37.059,179.895,5.236,148.937
C02388=1235.900,-71.081,-37.047,179.893,5.236,148.938
C02389=1235.905,-71.331,-37.034,179.891,5.236,148.939
C02390=1235.910,-71.580,-37.023,179.888,5.236,148.940
C02391=1235.915,-71.830,-37.011,179.886,5.235,148.940
C02392=1235.921,-72.080,-36.999,179.884,5.236,148.941
C02393=1235.925,-72.330,-36.988,179.881,5.235,148.942
C02394=1235.930,-72.579,-36.975,179.879,5.236,148.942
C02395=1235.936,-72.829,-36.963,179.876,5.235,148.943
C02396=1235.941,-73.079,-36.952,179.874,5.236,148.944
C02397=1235.947,-73.328,-36.941,179.871,5.235,148.945
C02398=1235.951,-73.578,-36.929,179.869,5.235,148.945
C02399=1235.957,-73.828,-36.917,179.867,5.235,148.946
C02400=1235.962,-74.098,-36.904,179.864,5.235,148.947
C02401=1235.967,-74.368,-36.891,179.861,5.235,148.948
C02402=1235.973,-74.638,-36.879,179.859,5.235,148.948
C02403=1235.979,-74.909,-36.867,179.856,5.235,148.949
C02404=1235.984,-75.159,-36.855,179.854,5.235,148.950
C02405=1235.989,-75.408,-36.843,179.851,5.235,148.951
C02406=1235.995,-75.657,-36.831,179.849,5.235,148.951
C02407=1235.999,-75.907,-36.820,179.847,5.235,148.952
C02408=1236.005,-76.157,-36.808,179.844,5.235,148.953
C02409=1236.010,-76.407,-36.796,179.842,5.235,148.953
C02410=1236.015,-76.656,-36.785,179.839,5.235,148.954
C02411=1236.020,-76.906,-36.773,179.837,5.235,148.955
C02412=1236.025,-77.156,-36.762,179.834,5.234,148.956
C02413=1236.031,-77.406,-36.750,179.832,5.235,148.956
C02414=1236.036,-77.655,-36.739,179.830,5.234,148.957
C02415=1236.041,-77.905,-36.727,179.828,5.235,148.958
C02416=1236.046,-78.154,-36.716,179.825,5.234,148.958
C02417=1236.051,-78.404,-36.704,179.823,5.235,148.959
C02418=1236.056,-78.654,-36.693,179.820,5.234,148.960
C02419=1236.062,-78.904,-36.681,179.818,5.234,148.961
C02420=1236.067,-79.153,-36.670,179.815,5.234,148.961
C02421=1236.072,-79.402,-36.658,179.813,5.234,148.962
C02422=1236.077,-79.652,-36.647,179.811,5.234,148.963
C02423=1236.082,-79.902,-36.635,179.809,5.234,148.963
C02424=1236.087,-80.152,-36.623,179.806,5.234,148.964
C02425=1236.092,-80.402,-36.611,179.804,5.234,148.965
C02426=1236.098,-80.651,-36.601,179.801,5.234,148.966
C02427=1236.103,-80.900,-36.589,179.799,5.234,148.966
C02428=1236.108,-81.150,-36.577,179.796,5.233,148.967
C02429=1236.113,-81.400,-36.565,179.794,5.234,148.968
C02430=1236.118,-81.650,-36.555,179.792,5.233,148.968
C02431=1236.124,-81.900,-36.543,179.790,5.234,148.969
C02432=1236.129,-82.149,-36.532,179.787,5.233,148.970
C02433=1236.134,-82.399,-36.521,179.785,5.234,148.971
C02434=1236.139,-82.649,-36.509,179.782,5.233,148.971
C02435=1236.144,-82.898,-36.498,179.779,5.234,148.972
C02436=1236.150,-83.148,-36.486,179.777,5.233,148.973
C02437=1236.155,-83.397,-36.475,179.775,5.234,148.974
C02438=1236.160,-83.647,-36.463,179.772,5.233,148.974
C02439=1236.165,-83.897,-36.452,179.770,5.234,148.975
C02440=1236.170,-84.147,-36.441,179.767,5.233,148.976
C02441=1236.176,-84.396,-36.430,179.765,5.233,148.976
C02442=1236.180,-84.646,-36.418,179.763,5.233,148.977
C02443=1236.186,-84.896,-36.406,179.760,5.233,148.978
C02444=1236.191,-85.145,-36.395,179.758,5.233,148.979
C02445=1236.196,-85.395,-36.385,179.756,5.233,148.979
C02446=1236.202,-85.645,-36.373,179.753,5.233,148.980
C02447=1236.206,-85.895,-36.362,179.751,5.233,148.981
C02448=1236.211,-86.144,-36.350,179.748,5.233,148.981
C02449=1236.217,-86.393,-36.339,179.746,5.233,148.982
C02450=1236.222,-86.644,-36.328,179.743,5.233,148.983
C02451=1236.227,-86.893,-36.317,179.741,5.233,148.984
C02452=1236.232,-87.143,-36.305,179.739,5.232,148.984
C02453=1236.237,-87.392,-36.294,179.737,5.233,148.985
C02454=1236.242,-87.642,-36.284,179.734,5.232,148.986
C02455=1236.248,-87.892,-36.272,179.732,5.233,148.986
C02456=1236.253,-88.142,-36.260,179.729,5.232,148.987
C02457=1236.258,-88.391,-36.250,179.727,5.233,148.988
C02458=1236.264,-88.641,-36.238,179.725,5.233,148.989
C02459=1236.268,-88.891,-36.227,179.722,5.232,148.989
C02460=1236.274,-89.140,-36.216,179.720,5.233,148.990
C02461=1236.279,-89.391,-36.205,179.718,5.232,148.991
C02462=1236.284,-89.640,-36.194,179.715,5.233,148.991
C02463=1236.289,-89.890,-36.182,179.713,5.232,148.992
C02464=1236.294,-90.139,-36.172,179.711,5.233,148.993
C02465=1236.300,-90.389,-36.160,179.708,5.232,148.993
C02466=1236.304,-90.639,-36.149,179.706,5.232,148.994
C02467=1236.310,-90.888,-36.139,179.703,5.232,148.995
C02468=1236.315,-91.138,-36.127,179.701,5.232,148.996
C02469=1236.320,-91.388,-36.116,179.698,5.232,148.996
C02470=1236.326,-91.638,-36.105,179.696,5.232,148.997
C02471=1236.330,-91.887,-36.094,179.694,5.232,148.998
C02472=1236.336,-92.137,-36.082,179.692,5.232,148.998
C02473=1236.341,-92.387,-36.072,179.689,5.232,148.999
C02474=1236.346,-92.636,-36.061,179.687,5.232,149.000
C02475=1236.351,-92.887,-36.050,179.684,5.232,149.001
C02476=1236.357,-93.136,-36.039,179.682,5.232,149.001
C02477=1236.362,-93.385,-36.027,179.679,5.231,149.002
C02478=1236.367,-93.636,-36.017,179.677,5.232,149.003
C02479=1236.372,-93.885,-36.006,179.675,5.231,149.003
C02480=1236.377,-94.135,-35.995,179.673,5.232,149.004
C02481=1236.383,-94.385,-35.983,179.670,5.232,149.005
C02482=1236.388,-94.634,-35.973,179.668,5.232,149.006
C02483=1236.393,-94.884,-35.962,179.666,5.232,149.006
C02484=1236.398,-95.133,-35.951,179.663,5.232,149.007
C02485=1236.403,-95.383,-35.940,179.661,5.232,149.008
C02486=1236.409,-95.633,-35.929,179.658,5.231,149.008
C02487=1236.414,-95.883,-35.918,179.656,5.232,149.009
C02488=1236.419,-96.132,-35.907,179.653,5.231,149.010
C02489=1236.424,-96.382,-35.897,179.651,5.232,149.011
C02490=1236.429,-96.631,-35.886,179.649,5.231,149.011
C02491=1236.434,-96.882,-35.875,179.647,5.232,149.012
C02492=1236.440,-97.131,-35.863,179.644,5.231,149.013
C02493=1236.445,-97.381,-35.853,179.642,5.231,149.013
C02494=1236.450,-97.630,-35.842,179.639,5.231,149.014
C02495=1236.455,-97.880,-35.831,179.637,5.231,149.015
C02496=1236.460,-98.130,-35.820,179.635,5.232,149.016
C02497=1236.466,-98.379,-35.810,179.632,5.231,149.016
C02498=1236.471,-98.630,-35.799,179.630,5.232,149.017
C02499=1236.476,-98.879,-35.788,179.628,5.231,149.018
C02500=1236.482,-99.129,-35.777,179.625,5.232,149.018
C02501=1236.486,-99.379,-35.766,179.623,5.231,149.019
C02502=1236.492,-99.628,-35.756,179.621,5.231,149.020
C02503=1236.497,-99.878,-35.744,179.618,5.231,149.021
C02504=1236.503,-100.148,-35.734,179.616,5.231,149.021
C02505=1236.508,-100.419,-35.722,179.613,5.231,149.022
C02506=1236.514,-100.690,-35.709,179.610,5.231,149.023
C02507=1236.520,-100.961,-35.699,179.608,5.231,149.024
C02508=1236.524,-101.211,-35.687,179.605,5.231,149.024
C02509=1236.529,-101.461,-35.677,179.603,5.231,149.025
C02510=1236.535,-101.710,-35.667,179.600,5.231,149.026
C02511=1236.540,-101.960,-35.655,179.598,5.231,149.027
C02512=1236.546,-102.210,-35.645,179.596,5.231,149.027
C02513=1236.551,-102.460,-35.634,179.594,5.231,149.028
C02514=1236.556,-102.709,-35.623,179.592,5.231,149.029
C02515=1236.561,-102.959,-35.613,179.589,5.231,149.029
C02516=1236.567,-103.209,-35.602,179.587,5.231,149.030
C02517=1236.571,-103.459,-35.591,179.584,5.231,149.031
C02518=1236.577,-103.708,-35.581,179.582,5.231,149.032
C02519=1236.582,-103.958,-35.570,179.579,5.231,149.032
C02520=1236.587,-104.207,-35.559,179.577,5.231,149.033
C02521=1236.592,-104.457,-35.549,179.575,5.231,149.034
C02522=1236.598,-104.707,-35.539,179.572,5.231,149.034
C02523=1236.603,-104.957,-35.528,179.570,5.231,149.035
C02524=1236.608,-105.206,-35.517,179.568,5.231,149.036
C02525=1236.613,-105.456,-35.506,179.566,5.231,149.037
C02526=1236.619,-105.706,-35.496,179.563,5.230,149.037
C02527=1236.624,-105.956,-35.486,179.561,5.231,149.038
C02528=1236.629,-106.205,-35.475,179.559,5.230,149.038
C02529=1236.634,-106.455,-35.464,179.557,5.231,149.039
C02530=1236.639,-106.705,-35.455,179.554,5.230,149.040
C02531=1236.644,-106.955,-35.444,179.552,5.231,149.041
C02532=1236.649,-107.204,-35.433,179.549,5.230,149.041
C02533=1236.654,-107.454,-35.423,179.547,5.231,149.042
C02534=1236.660,-107.704,-35.412,179.544,5.230,149.043
C02535=1236.665,-107.954,-35.402,179.542,5.230,149.043
C02536=1236.670,-108.203,-35.392,179.540,5.231,149.044
C02537=1236.675,-108.453,-35.380,179.537,5.230,149.045
C02538=1236.681,-108.703,-35.370,179.535,5.231,149.046
C02539=1236.686,-108.952,-35.360,179.533,5.230,149.046
C02540=1236.691,-109.202,-35.349,179.531,5.231,149.047
C02541=1236.697,-109.452,-35.339,179.528,5.230,149.048
C02542=1236.702,-109.702,-35.328,179.526,5.231,149.048
C02543=1236.707,-109.951,-35.319,179.523,5.230,149.049
C02544=1236.711,-110.201,-35.308,179.521,5.230,149.050
C02545=1236.717,-110.451,-35.297,179.518,5.230,149.051
C02546=1236.723,-110.700,-35.287,179.516,5.230,149.051
C02547=1236.728,-110.950,-35.277,179.514,5.231,149.052
C02548=1236.733,-111.200,-35.266,179.511,5.230,149.053
C02549=1236.738,-111.450,-35.256,179.509,5.231,149.053
C02550=1236.744,-111.700,-35.246,179.507,5.230,149.054
C02551=1236.749,-111.950,-35.235,179.505,5.231,149.055
C02552=1236.754,-112.199,-35.225,179.502,5.230,149.055
C02553=1236.759,-112.449,-35.215,179.500,5.230,149.056
C02554=1236.764,-112.698,-35.204,179.498,5.230,149.057
C02555=1236.770,-112.948,-35.194,179.496,5.230,149.057
C02556=1236.775,-113.197,-35.183,179.493,5.230,149.058
C02557=1236.780,-113.448,-35.173,179.491,5.230,149.059
C02558=1236.785,-113.697,-35.163,179.489,5.230,149.060
C02559=1236.790,-113.947,-35.153,179.486,5.230,149.060
C02560=1236.796,-114.197,-35.142,179.484,5.230,149.061
C02561=1236.801,-114.446,-35.132,179.481,5.230,149.062
C02562=1236.806,-114.696,-35.122,179.479,5.230,149.062
C02563=1236.811,-114.946,-35.112,179.476,5.230,149.063
C02564=1236.817,-115.195,-35.102,179.474,5.230,149.064
C02565=1236.822,-115.445,-35.091,179.472,5.230,149.065
C02566=1236.827,-115.695,-35.081,179.470,5.230,149.065
C02567=1236.832,-115.945,-35.071,179.468,5.230,149.066
C02568=1236.837,-116.194,-35.061,179.465,5.230,149.067
C02569=1236.843,-116.444,-35.051,179.463,5.230,149.067
C02570=1236.848,-116.694,-35.040,179.461,5.230,149.068
C02571=1236.853,-116.944,-35.030,179.458,5.230,149.069
C02572=1236.858,-117.193,-35.020,179.456,5.230,149.069
C02573=1236.863,-117.443,-35.010,179.454,5.230,149.070
C02574=1236.869,-117.693,-35.000,179.451,5.229,149.071
C02575=1236.875,-117.943,-34.990,179.449,5.230,149.072
C02576=1236.879,-118.193,-34.980,179.447,5.230,149.072
C02577=1236.885,-118.442,-34.970,179.444,5.230,149.073
C02578=1236.890,-118.692,-34.960,179.442,5.230,149.074
C02579=1236.895,-118.942,-34.949,179.439,5.230,149.074
C02580=1236.900,-119.191,-34.939,179.437,5.230,149.075
C02581=1236.906,-119.441,-34.929,179.435,5.230,149.076
C02582=1236.911,-119.691,-34.919,179.432,5.230,149.077
C02583=1236.915,-119.940,-34.909,179.430,5.229,149.077
C02584=1236.921,-120.191,-34.900,179.428,5.230,149.078
C02585=1236.927,-120.440,-34.889,179.426,5.230,149.079
C02586=1236.931,-120.690,-34.879,179.423,5.229,149.079
C02587=1236.937,-120.940,-34.869,179.421,5.230,149.080
C02588=1236.942,-121.189,-34.859,179.419,5.229,149.081
C02589=1236.947,-121.439,-34.849,179.417,5.230,149.081
C02590=1236.953,-121.689,-34.839,179.414,5.229,149.082
C02591=1236.958,-121.939,-34.829,179.412,5.230,149.083
C02592=1236.963,-122.188,-34.820,179.409,5.229,149.084
C02593=1236.968,-122.438,-34.809,179.407,5.230,149.084
C02594=1236.974,-122.688,-34.799,179.405,5.230,149.085
C02595=1236.979,-122.938,-34.790,179.402,5.230,149.086
C02596=1236.984,-123.187,-34.780,179.401,5.230,149.086
C02597=1236.989,-123.438,-34.769,179.398,5.229,149.087
C02598=1236.994,-123.687,-34.760,179.396,5.230,149.088
C02599=1237.000,-123.936,-34.749,179.393,5.229,149.088
C02600=1237.006,-124.186,-34.740,179.391,5.229,149.089
C02601=1237.010,-124.436,-34.730,179.389,5.230,149.090
C02602=1237.016,-124.686,-34.720,179.386,5.229,149.090
C02603=1237.020,-124.935,-34.710,179.384,5.230,149.091
C02604=1237.026,-125.185,-34.701,179.382,5.229,149.092
C02605=1237.031,-125.436,-34.690,179.379,5.230,149.093
C02606=1237.036,-125.685,-34.680,179.377,5.229,149.093
C02607=1237.042,-125.935,-34.671,179.375,5.229,149.094
C02608=1236.621,-125.945,-34.706,179.371,5.233,149.096
C02609=1236.615,-125.695,-34.715,179.373,5.232,149.095
C02610=1236.609,-125.446,-34.726,179.375,5.233,149.095
C02611=1236.604,-125.196,-34.735,179.378,5.232,149.094
C02612=1236.599,-124.946,-34.745,179.380,5.233,149.093
C02613=1236.594,-124.696,-34.755,179.382,5.233,149.093
C02614=1236.589,-124.447,-34.765,179.384,5.233,149.092
C02615=1236.583,-124.197,-34.775,179.387,5.233,149.091
C02616=1236.578,-123.947,-34.784,179.389,5.233,149.090
C02617=1236.573,-123.697,-34.795,179.391,5.233,149.090
C02618=1236.567,-123.448,-34.805,179.393,5.233,149.089
C02619=1236.562,-123.198,-34.814,179.396,5.233,149.088
C02620=1236.557,-122.949,-34.825,179.398,5.233,149.088
C02621=1236.552,-122.698,-34.834,179.401,5.233,149.087
C02622=1236.547,-122.449,-34.844,179.403,5.233,149.086
C02623=1236.541,-122.199,-34.854,179.405,5.233,149.086
C02624=1236.536,-121.950,-34.864,179.407,5.233,149.085
C02625=1236.531,-121.700,-34.875,179.409,5.233,149.084
C02626=1236.525,-121.450,-34.884,179.412,5.233,149.083
C02627=1236.521,-121.200,-34.894,179.414,5.233,149.083
C02628=1236.516,-120.950,-34.904,179.417,5.233,149.082
C02629=1236.510,-120.701,-34.914,179.419,5.233,149.081
C02630=1236.505,-120.451,-34.924,179.422,5.233,149.081
C02631=1236.499,-120.202,-34.934,179.424,5.233,149.080
C02632=1236.494,-119.951,-34.944,179.426,5.233,149.079
C02633=1236.489,-119.702,-34.954,179.429,5.233,149.078
C02634=1236.484,-119.452,-34.964,179.431,5.233,149.078
C02635=1236.479,-119.202,-34.974,179.433,5.234,149.077
C02636=1236.473,-118.952,-34.985,179.435,5.233,149.077
C02637=1236.468,-118.703,-34.994,179.438,5.234,149.076
C02638=1236.463,-118.453,-35.005,179.440,5.233,149.075
C02639=1236.458,-118.203,-35.015,179.442,5.234,149.074
C02640=1236.452,-117.953,-35.024,179.444,5.233,149.074
C02641=1236.447,-117.703,-35.035,179.447,5.233,149.073
C02642=1236.442,-117.454,-35.045,179.449,5.233,149.072
C02643=1236.436,-117.204,-35.055,179.451,5.233,149.072
C02644=1236.432,-116.954,-35.065,179.454,5.233,149.071
C02645=1236.426,-116.705,-35.075,179.456,5.233,149.070
C02646=1236.421,-116.455,-35.085,179.459,5.234,149.069
C02647=1236.416,-116.205,-35.096,179.461,5.233,149.069
C02648=1236.411,-115.956,-35.106,179.464,5.234,149.068
C02649=1236.405,-115.706,-35.116,179.465,5.234,149.067
C02650=1236.400,-115.456,-35.126,179.467,5.233,149.067
C02651=1236.395,-115.206,-35.137,179.470,5.234,149.066
C02652=1236.389,-114.957,-35.147,179.472,5.233,149.065
C02653=1236.385,-114.707,-35.157,179.475,5.234,149.065
C02654=1236.379,-114.457,-35.167,179.477,5.233,149.064
C02655=1236.374,-114.208,-35.177,179.479,5.234,149.063
C02656=1236.369,-113.958,-35.188,179.482,5.233,149.062
C02657=1236.363,-113.708,-35.198,179.484,5.234,149.062
C02658=1236.359,-113.458,-35.208,179.486,5.234,149.061
C02659=1236.353,-113.209,-35.218,179.488,5.233,149.060
C02660=1236.348,-112.959,-35.228,179.491,5.234,149.060
C02661=1236.343,-112.709,-35.239,179.493,5.233,149.059
C02662=1236.337,-112.459,-35.249,179.496,5.234,149.058
C02663=1236.332,-112.209,-35.260,179.498,5.233,149.057
C02664=1236.327,-111.960,-35.269,179.501,5.234,149.057
C02665=1236.322,-111.710,-35.280,179.503,5.233,149.056
C02666=1236.317,-111.461,-35.291,179.505,5.234,149.055
C02667=1236.311,-111.211,-35.301,179.507,5.234,149.055
C02668=1236.306,-110.961,-35.312,179.510,5.234,149.054
C02669=1236.301,-110.711,-35.322,179.512,5.234,149.053
C02670=1236.295,-110.462,-35.332,179.514,5.234,149.053
C02671=1236.290,-110.211,-35.343,179.517,5.234,149.052
C02672=1236.285,-109.962,-35.352,179.519,5.234,149.051
C02673=1236.280,-109.712,-35.363,179.521,5.234,149.051
C02674=1236.275,-109.462,-35.373,179.523,5.234,149.050
C02675=1236.270,-109.213,-35.384,179.526,5.234,149.049
C02676=1236.264,-108.963,-35.394,179.528,5.234,149.048
C02677=1236.259,-108.714,-35.405,179.531,5.234,149.048
C02678=1236.254,-108.463,-35.415,179.533,5.234,149.047
C02679=1236.248,-108.214,-35.425,179.536,5.234,149.046
C02680=1236.243,-107.964,-35.436,179.538,5.234,149.046
C02681=1236.238,-107.715,-35.447,179.540,5.234,149.045
C02682=1236.233,-107.464,-35.458,179.543,5.234,149.044
C02683=1236.227,-107.215,-35.468,179.545,5.234,149.043
C02684=1236.223,-106.965,-35.478,179.547,5.234,149.043
C02685=1236.217,-106.715,-35.488,179.549,5.234,149.042
C02686=1236.213,-106.466,-35.499,179.552,5.234,149.041
C02687=1236.207,-106.216,-35.509,179.554,5.234,149.041
C02688=1236.202,-105.966,-35.520,179.557,5.234,149.040
C02689=1236.197,-105.716,-35.530,179.559,5.234,149.039
C02690=1236.191,-105.468,-35.541,179.562,5.234,149.038
C02691=1236.186,-105.217,-35.552,179.563,5.234,149.038
C02692=1236.181,-104.968,-35.562,179.565,5.234,149.037
C02693=1236.176,-104.718,-35.573,179.568,5.234,149.036
C02694=1236.170,-104.469,-35.583,179.570,5.234,149.036
C02695=1236.165,-104.218,-35.594,179.573,5.235,149.035
C02696=1236.160,-103.969,-35.604,179.575,5.234,149.034
C02697=1236.155,-103.719,-35.616,179.578,5.235,149.034
C02698=1236.149,-103.470,-35.626,179.580,5.234,149.033
C02699=1236.144,-103.219,-35.636,179.582,5.235,149.032
C02700=1236.139,-102.969,-35.647,179.584,5.234,149.031
C02701=1236.134,-102.720,-35.658,179.587,5.235,149.031
C02702=1236.129,-102.470,-35.668,179.589,5.234,149.030
C02703=1236.124,-102.220,-35.679,179.592,5.235,149.029
C02704=1236.119,-101.971,-35.690,179.594,5.235,149.029
C02705=1236.113,-101.721,-35.700,179.596,5.234,149.028
C02706=1236.108,-101.471,-35.711,179.599,5.235,149.027
C02707=1236.103,-101.222,-35.722,179.601,5.234,149.026
C02708=1236.098,-100.972,-35.732,179.603,5.235,149.026
C02709=1236.092,-100.701,-35.744,179.606,5.234,149.025
C02710=1236.086,-100.430,-35.756,179.608,5.235,149.024
C02711=1236.081,-100.159,-35.767,179.611,5.235,149.023
C02712=1236.075,-99.888,-35.779,179.614,5.234,149.023
C02713=1236.070,-99.639,-35.790,179.616,5.235,149.022
C02714=1236.065,-99.389,-35.801,179.618,5.235,149.021
C02715=1236.060,-99.140,-35.811,179.621,5.235,149.021
C02716=1236.055,-98.889,-35.822,179.623,5.235,149.020
C02717=1236.049,-98.640,-35.833,179.626,5.235,149.019
C02718=1236.044,-98.390,-35.843,179.628,5.235,149.018
C02719=1236.039,-98.140,-35.855,179.630,5.234,149.018
C02720=1236.033,-97.891,-35.865,179.633,5.235,149.017
C02721=1236.029,-97.641,-35.877,179.635,5.235,149.016
C02722=1236.023,-97.392,-35.887,179.637,5.235,149.016
C02723=1236.018,-97.142,-35.898,179.639,5.235,149.015
C02724=1236.013,-96.892,-35.909,179.642,5.235,149.014
C02725=1236.008,-96.643,-35.920,179.644,5.235,149.013
C02726=1236.002,-96.392,-35.931,179.647,5.235,149.013
C02727=1235.997,-96.143,-35.942,179.649,5.235,149.012
C02728=1235.992,-95.893,-35.952,179.652,5.235,149.011
C02729=1235.987,-95.643,-35.964,179.654,5.235,149.011
C02730=1235.982,-95.394,-35.974,179.656,5.235,149.010
C02731=1235.977,-95.144,-35.985,179.659,5.235,149.009
C02732=1235.971,-94.894,-35.996,179.661,5.235,149.008
C02733=1235.966,-94.645,-36.007,179.663,5.235,149.008
C02734=1235.961,-94.395,-36.018,179.666,5.236,149.007
C02735=1235.956,-94.146,-36.029,179.668,5.235,149.006
C02736=1235.951,-93.895,-36.039,179.670,5.235,149.006
C02737=1235.945,-93.645,-36.051,179.673,5.235,149.005
C02738=1235.940,-93.396,-36.061,179.675,5.235,149.004
C02739=1235.935,-93.146,-36.073,179.678,5.235,149.003
C02740=1235.930,-92.897,-36.084,179.680,5.235,149.003
C02741=1235.924,-92.647,-36.095,179.682,5.235,149.002
C02742=1235.919,-92.397,-36.106,179.684,5.235,149.001
C02743=1235.914,-92.148,-36.116,179.687,5.236,149.001
C02744=1235.909,-91.898,-36.128,179.689,5.235,149.000
C02745=1235.904,-91.648,-36.139,179.692,5.236,148.999
C02746=1235.898,-91.399,-36.150,179.694,5.235,148.998
C02747=1235.893,-91.149,-36.161,179.697,5.236,148.998
C02748=1235.888,-90.899,-36.172,179.699,5.235,148.997
C02749=1235.883,-90.649,-36.183,179.701,5.236,148.996
C02750=1235.877,-90.400,-36.194,179.704,5.236,148.996
C02751=1235.873,-90.150,-36.206,179.706,5.236,148.995
C02752=1235.868,-89.900,-36.216,179.708,5.236,148.994
C02753=1235.862,-89.651,-36.228,179.711,5.236,148.993
C02754=1235.857,-89.401,-36.239,179.713,5.236,148.993
C02755=1235.852,-89.151,-36.250,179.716,5.236,148.992
C02756=1235.846,-88.902,-36.261,179.718,5.236,148.991
C02757=1235.841,-88.652,-36.272,179.720,5.236,148.991
C02758=1235.836,-88.402,-36.283,179.723,5.236,148.990
C02759=1235.832,-88.152,-36.294,179.725,5.236,148.989
C02760=1235.826,-87.903,-36.306,179.727,5.236,148.988
C02761=1235.821,-87.653,-36.317,179.729,5.236,148.988
C02762=1235.816,-87.403,-36.328,179.732,5.236,148.987
C02763=1235.810,-87.154,-36.339,179.734,5.236,148.986
C02764=1235.805,-86.904,-36.350,179.737,5.236,148.986
C02765=1235.800,-86.654,-36.362,179.739,5.236,148.985
C02766=1235.795,-86.404,-36.373,179.742,5.236,148.984
C02767=1235.789,-86.155,-36.384,179.744,5.236,148.984
C02768=1235.785,-85.905,-36.395,179.746,5.237,148.983
C02769=1235.779,-85.655,-36.407,179.749,5.236,148.982
C02770=1235.775,-85.406,-36.418,179.751,5.237,148.981
C02771=1235.768,-85.156,-36.429,179.753,5.236,148.981
C02772=1235.764,-84.906,-36.440,179.756,5.237,148.980
C02773=1235.759,-84.657,-36.452,179.758,5.236,148.979
C02774=1235.753,-84.407,-36.464,179.761,5.237,148.979
C02775=1235.748,-84.158,-36.474,179.763,5.237,148.978
C02776=1235.743,-83.908,-36.485,179.765,5.237,148.977
C02777=1235.738,-83.658,-36.497,179.768,5.237,148.976
C02778=1235.733,-83.408,-36.508,179.770,5.237,148.976
C02779=1235.728,-83.158,-36.520,179.772,5.237,148.975
C02780=1235.722,-82.909,-36.531,179.775,5.237,148.974
C02781=1235.717,-82.659,-36.543,179.777,5.237,148.974
C02782=1235.712,-82.410,-36.554,179.780,5.237,148.973
C02783=1235.708,-82.160,-36.565,179.782,5.237,148.972
C02784=1235.702,-81.909,-36.577,179.785,5.237,148.971
C02785=1235.697,-81.661,-36.588,179.787,5.237,148.971
C02786=1235.691,-81.411,-36.599,179.789,5.238,148.970
C02787=1235.686,-81.161,-36.611,179.791,5.237,148.969
C02788=1235.681,-80.911,-36.623,179.794,5.238,148.969
C02789=1235.676,-80.661,-36.634,179.796,5.237,148.968
C02790=1235.670,-80.412,-36.645,179.799,5.238,148.967
C02791=1235.666,-80.163,-36.657,179.801,5.237,148.966
C02792=1235.661,-79.913,-36.668,179.804,5.238,148.966
C02793=1235.655,-79.663,-36.680,179.806,5.237,148.965
C02794=1235.651,-79.413,-36.691,179.809,5.238,148.964
C02795=1235.645,-79.163,-36.703,179.811,5.237,148.963
C02796=1235.640,-78.914,-36.714,179.814,5.238,148.963
C02797=1235.635,-78.665,-36.726,179.816,5.237,148.962
C02798=1235.630,-78.415,-36.737,179.818,5.238,148.961
C02799=1235.624,-78.165,-36.749,179.820,5.238,148.961
C02800=1235.619,-77.915,-36.761,179.823,5.238,148.960
C02801=1235.614,-77.665,-36.772,179.825,5.238,148.959
C02802=1235.608,-77.416,-36.784,179.828,5.238,148.958
C02803=1235.604,-77.167,-36.795,179.830,5.238,148.958
C02804=1235.598,-76.917,-36.807,179.833,5.238,148.957
C02805=1235.593,-76.667,-36.818,179.835,5.238,148.956
C02806=1235.588,-76.417,-36.830,179.837,5.238,148.956
C02807=1235.583,-76.167,-36.841,179.840,5.238,148.955
C02808=1235.578,-75.917,-36.853,179.842,5.239,148.954
C02809=1235.573,-75.669,-36.864,179.844,5.238,148.953
C02810=1235.567,-75.419,-36.876,179.847,5.239,148.953
C02811=1235.562,-75.169,-36.888,179.849,5.238,148.952
C02812=1235.557,-74.919,-36.899,179.852,5.239,148.951
C02813=1235.552,-74.649,-36.912,179.854,5.239,148.951
C02814=1235.546,-74.379,-36.925,179.857,5.239,148.950
C02815=1235.540,-74.108,-36.937,179.859,5.238,148.949
C02816=1235.535,-73.838,-36.950,179.862,5.239,148.948
C02817=1235.530,-73.588,-36.962,179.864,5.239,148.948
C02818=1235.524,-73.339,-36.973,179.866,5.239,148.947
C02819=1235.519,-73.090,-36.985,179.869,5.239,148.946
C02820=1235.514,-72.840,-36.997,179.871,5.239,148.945
C02821=1235.509,-72.590,-37.009,179.874,5.239,148.945
C02822=1235.504,-72.340,-37.021,179.877,5.239,148.944
C02823=1235.498,-72.090,-37.032,179.879,5.239,148.943
C02824=1235.493,-71.840,-37.044,179.881,5.239,148.942
C02825=1235.488,-71.591,-37.056,179.884,5.239,148.942
C02826=1235.483,-71.341,-37.068,179.886,5.239,148.941
C02827=1235.478,-71.092,-37.079,179.889,5.239,148.940
C02828=1235.473,-70.842,-37.091,179.891,5.239,148.940
C02829=1235.467,-70.592,-37.103,179.893,5.240,148.939
C02830=1235.463,-70.343,-37.115,179.896,5.239,148.938
C02831=1235.458,-70.093,-37.127,179.898,5.240,148.937
C02832=1235.452,-69.843,-37.139,179.900,5.239,148.937
C02833=1235.447,-69.594,-37.150,179.903,5.240,148.936
C02834=1235.442,-69.345,-37.163,179.905,5.240,148.935
C02835=1235.436,-69.095,-37.174,179.908,5.240,148.935
C02836=1235.432,-68.845,-37.186,179.910,5.240,148.934
C02837=1235.426,-68.595,-37.198,179.913,5.240,148.933
C02838=1235.421,-68.346,-37.210,179.915,5.240,148.932
C02839=1235.416,-68.096,-37.222,179.917,5.240,148.932
C02840=1235.411,-67.846,-37.233,179.919,5.240,148.931
C02841=1235.405,-67.596,-37.245,179.922,5.240,148.930
C02842=1235.400,-67.347,-37.258,179.924,5.240,148.930
C02843=1235.396,-67.097,-37.269,179.927,5.241,148.929
C02844=1235.390,-66.847,-37.281,179.929,5.240,148.928
C02845=1235.385,-66.598,-37.294,179.932,5.240,148.927
C02846=1235.380,-66.348,-37.306,179.935,5.241,148.927
C02847=1235.375,-66.099,-37.317,179.937,5.241,148.926
C02848=1235.370,-65.849,-37.329,179.939,5.241,148.925
C02849=1235.364,-65.599,-37.341,179.942,5.241,148.924
C02850=1235.359,-65.349,-37.353,179.944,5.241,148.924
C02851=1235.354,-65.100,-37.366,179.946,5.241,148.923
C02852=1235.349,-64.850,-37.377,179.949,5.241,148.922
C02853=1235.344,-64.600,-37.389,179.951,5.241,148.922
C02854=1235.339,-64.351,-37.402,179.954,5.241,148.921
C02855=1235.333,-64.101,-37.413,179.956,5.241,148.920
C02856=1235.329,-63.852,-37.425,179.958,5.242,148.920
C02857=1235.324,-63.602,-37.438,179.961,5.241,148.919
C02858=1235.319,-63.352,-37.450,179.963,5.242,148.918
C02859=1235.313,-63.102,-37.462,179.965,5.241,148.917
C02860=1235.308,-62.852,-37.474,179.968,5.242,148.917
C02861=1235.303,-62.603,-37.487,179.970,5.242,148.916
C02862=1235.298,-62.353,-37.498,179.973,5.242,148.915
C02863=1235.293,-62.104,-37.511,179.975,5.242,148.915
C02864=1235.288,-61.854,-37.522,179.978,5.242,148.914
C02865=1235.282,-61.605,-37.535,179.980,5.241,148.913
C02866=1235.277,-61.355,-37.547,179.983,5.242,148.912
C02867=1235.272,-61.106,-37.560,179.985,5.242,148.912
C02868=1235.267,-60.856,-37.571,179.988,5.242,148.911
C02869=1235.262,-60.607,-37.583,179.990,5.243,148.910
C02870=1235.257,-60.357,-37.595,179.992,5.242,148.909
C02871=1235.252,-60.107,-37.608,179.995,5.243,148.909
C02872=1235.247,-59.857,-37.620,179.997,5.242,148.908
C02873=1235.242,-59.607,-37.633,180.000,5.243,148.907
C02874=1235.236,-59.358,-37.645,-179.998,5.243,148.907
C02875=1235.231,-59.108,-37.657,-179.996,5.243,148.906
C02876=1235.226,-58.858,-37.669,-179.993,5.243,148.905
C02877=1235.221,-58.609,-37.681,-179.991,5.243,148.904
C02878=1235.216,-58.359,-37.693,-179.989,5.243,148.904
C02879=1235.211,-58.110,-37.706,-179.986,5.243,148.903
C02880=1235.205,-57.860,-37.718,-179.983,5.244,148.902
C02881=1235.201,-57.610,-37.730,-179.981,5.243,148.902
C02882=1235.196,-57.361,-37.743,-179.979,5.244,148.901
C02883=1235.190,-57.111,-37.755,-179.976,5.243,148.900
C02884=1235.185,-56.861,-37.768,-179.973,5.244,148.899
C02885=1235.180,-56.612,-37.779,-179.971,5.243,148.899
C02886=1235.175,-56.362,-37.792,-179.969,5.244,148.898
C02887=1235.169,-56.113,-37.805,-179.967,5.244,148.897
C02888=1235.165,-55.862,-37.817,-179.964,5.244,148.897
C02889=1235.159,-55.613,-37.830,-179.962,5.244,148.896
C02890=1235.154,-55.364,-37.842,-179.959,5.244,148.895
C02891=1235.149,-55.114,-37.854,-179.957,5.244,148.894
C02892=1235.144,-54.864,-37.867,-179.954,5.244,148.894
C02893=1235.138,-54.614,-37.878,-179.952,5.245,148.893
C02894=1235.134,-54.364,-37.891,-179.950,5.245,148.892
C02895=1235.129,-54.115,-37.904,-179.947,5.245,148.892
C02896=1235.124,-53.866,-37.917,-179.945,5.245,148.891
C02897=1235.118,-53.616,-37.929,-179.942,5.245,148.890
C02898=1235.113,-53.367,-37.941,-179.940,5.245,148.889
C02899=1235.108,-53.117,-37.954,-179.937,5.245,148.889
C02900=1235.103,-52.867,-37.966,-179.935,5.245,148.888
C02901=1235.098,-52.617,-37.979,-179.932,5.245,148.887
C02902=1235.093,-52.368,-37.991,-179.930,5.245,148.886
C02903=1235.088,-52.119,-38.004,-179.927,5.245,148.886
C02904=1235.083,-51.868,-38.016,-179.925,5.246,148.885
C02905=1235.078,-51.619,-38.029,-179.923,5.245,148.884
C02906=1235.073,-51.369,-38.041,-179.920,5.246,148.884
C02907=1235.067,-51.120,-38.054,-179.918,5.246,148.883
C02908=1235.062,-50.870,-38.066,-179.915,5.246,148.882
C02909=1235.058,-50.620,-38.079,-179.913,5.246,148.881
C02910=1235.052,-50.371,-38.091,-179.910,5.246,148.881
C02911=1235.047,-50.121,-38.104,-179.908,5.246,148.880
C02912=1235.042,-49.872,-38.116,-179.906,5.246,148.879
C02913=1235.037,-49.622,-38.128,-179.903,5.247,148.879
C02914=1235.031,-49.372,-38.142,-179.901,5.247,148.878
C02915=1235.026,-49.123,-38.155,-179.898,5.247,148.877
C02916=1235.021,-48.873,-38.167,-179.896,5.246,148.876
C02917=1235.016,-48.603,-38.181,-179.893,5.247,148.876
C02918=1235.011,-48.333,-38.194,-179.890,5.247,148.875
C02919=1235.005,-48.064,-38.208,-179.888,5.247,148.874
C02920=1235.000,-47.794,-38.221,-179.885,5.247,148.873
C02921=1234.994,-47.545,-38.234,-179.882,5.248,148.873
C02922=1234.989,-47.295,-38.247,-179.880,5.247,148.872
C02923=1234.984,-47.045,-38.260,-179.878,5.248,148.871
C02924=1234.979,-46.796,-38.273,-179.876,5.248,148.870
C02925=1234.974,-46.546,-38.285,-179.873,5.248,148.870
C02926=1234.968,-46.297,-38.297,-179.871,5.248,148.869
C02927=1234.964,-46.047,-38.310,-179.868,5.248,148.868
C02928=1234.959,-45.797,-38.323,-179.866,5.249,148.868
C02929=1234.953,-45.548,-38.336,-179.863,5.248,148.867
C02930=1234.948,-45.298,-38.349,-179.861,5.249,148.866
C02931=1234.943,-45.048,-38.362,-179.859,5.249,148.866
C02932=1234.938,-44.799,-38.374,-179.856,5.249,148.865
C02933=1234.934,-44.549,-38.387,-179.853,5.248,148.864
C02934=1234.928,-44.299,-38.400,-179.851,5.249,148.863
C02935=1234.923,-44.050,-38.413,-179.849,5.249,148.863
C02936=1234.917,-43.801,-38.426,-179.846,5.249,148.862
C02937=1234.913,-43.551,-38.439,-179.843,5.250,148.861
C02938=1234.907,-43.301,-38.452,-179.841,5.249,148.860
C02939=1234.902,-43.052,-38.464,-179.839,5.250,148.860
C02940=1234.897,-42.802,-38.477,-179.837,5.249,148.859
C02941=1234.892,-42.552,-38.490,-179.834,5.250,148.858
C02942=1234.887,-42.303,-38.502,-179.832,5.250,148.858
C02943=1234.882,-42.053,-38.516,-179.829,5.250,148.857
C02944=1234.877,-41.803,-38.529,-179.826,5.251,148.856
C02945=1234.872,-41.554,-38.541,-179.824,5.250,148.856
C02946=1234.867,-41.304,-38.554,-179.822,5.251,148.855
C02947=1234.861,-41.054,-38.567,-179.820,5.250,148.854
C02948=1234.856,-40.805,-38.580,-179.816,5.251,148.853
C02949=1234.852,-40.555,-38.593,-179.814,5.251,148.852
C02950=1234.846,-40.305,-38.606,-179.812,5.251,148.852
C02951=1234.841,-40.055,-38.619,-179.809,5.251,148.851
C02952=1234.836,-39.806,-38.632,-179.807,5.251,148.850
C02953=1234.831,-39.557,-38.645,-179.804,5.251,148.850
C02954=1234.826,-39.307,-38.659,-179.802,5.251,148.849
C02955=1234.821,-39.058,-38.671,-179.800,5.252,148.848
C02956=1234.816,-38.808,-38.684,-179.797,5.252,148.848
C02957=1234.811,-38.558,-38.697,-179.795,5.252,148.847
C02958=1234.805,-38.309,-38.710,-179.792,5.252,148.846
C02959=1234.801,-38.059,-38.723,-179.790,5.252,148.845
C02960=1234.795,-37.809,-38.736,-179.787,5.253,148.845
C02961=1234.790,-37.560,-38.749,-179.785,5.253,148.844
C02962=1234.786,-37.310,-38.762,-179.783,5.253,148.843
C02963=1234.780,-37.061,-38.776,-179.780,5.253,148.843
C02964=1234.775,-36.811,-38.789,-179.777,5.253,148.842
C02965=1234.769,-36.561,-38.802,-179.775,5.253,148.841
C02966=1234.764,-36.312,-38.814,-179.773,5.253,148.840
C02967=1234.760,-36.062,-38.828,-179.770,5.253,148.840
C02968=1234.754,-35.813,-38.841,-179.767,5.254,148.839
C02969=1234.750,-35.563,-38.854,-179.765,5.253,148.838
C02970=1234.744,-35.313,-38.867,-179.763,5.254,148.838
C02971=1234.739,-35.064,-38.881,-179.761,5.254,148.837
C02972=1234.735,-34.814,-38.894,-179.758,5.254,148.836
C02973=1234.729,-34.565,-38.907,-179.755,5.255,148.835
C02974=1234.724,-34.315,-38.920,-179.753,5.254,148.835
C02975=1234.719,-34.066,-38.934,-179.750,5.255,148.834
C02976=1234.714,-33.816,-38.947,-179.748,5.254,148.833
C02977=1234.709,-33.566,-38.959,-179.746,5.255,148.833
C02978=1234.704,-33.316,-38.973,-179.743,5.256,148.832
C02979=1234.699,-33.067,-38.986,-179.741,5.255,148.831
C02980=1234.693,-32.818,-38.999,-179.738,5.255,148.830
C02981=1234.688,-32.568,-39.012,-179.736,5.255,148.830
C02982=1234.683,-32.319,-39.026,-179.733,5.256,148.829
C02983=1234.678,-32.069,-39.039,-179.730,5.256,148.828
C02984=1234.673,-31.819,-39.052,-179.728,5.256,148.828
C02985=1234.668,-31.570,-39.066,-179.726,5.256,148.827
C02986=1234.662,-31.320,-39.079,-179.724,5.256,148.826
C02987=1234.658,-31.070,-39.092,-179.721,5.256,148.825
C02988=1234.652,-30.821,-39.106,-179.718,5.257,148.825
C02989=1234.648,-30.571,-39.119,-179.716,5.257,148.824
C02990=1234.643,-30.322,-39.132,-179.713,5.257,148.823
C02991=1234.638,-30.072,-39.146,-179.711,5.257,148.823
C02992=1234.633,-29.823,-39.159,-179.709,5.257,148.822
C02993=1234.627,-29.572,-39.172,-179.706,5.258,148.821
C02994=1234.622,-29.323,-39.186,-179.704,5.258,148.821
C02995=1234.617,-29.073,-39.199,-179.701,5.258,148.820
C02996=1234.612,-28.824,-39.213,-179.699,5.257,148.819
C02997=1234.607,-28.574,-39.226,-179.696,5.258,148.818
C02998=1234.602,-28.325,-39.240,-179.693,5.258,148.818
C02999=1234.597,-28.075,-39.253,-179.691,5.258,148.817
C03000=1234.591,-27.826,-39.266,-179.689,5.259,148.816
C03001=1234.587,-27.576,-39.280,-179.686,5.259,148.815
C03002=1234.582,-27.326,-39.293,-179.684,5.259,148.815
C03003=1234.577,-27.077,-39.307,-179.681,5.259,148.814
C03004=1234.572,-26.827,-39.320,-179.679,5.259,148.813
C03005=1234.566,-26.578,-39.334,-179.677,5.260,148.813
C03006=1234.562,-26.328,-39.347,-179.674,5.260,148.812
C03007=1234.556,-26.079,-39.361,-179.672,5.260,148.811
C03008=1234.552,-25.829,-39.374,-179.669,5.260,148.811
C03009=1234.546,-25.580,-39.388,-179.667,5.260,148.810
C03010=1234.542,-25.330,-39.401,-179.664,5.260,148.809
C03011=1234.537,-25.080,-39.415,-179.662,5.261,148.808
C03012=1234.531,-24.830,-39.428,-179.659,5.260,148.808
C03013=1234.526,-24.581,-39.442,-179.657,5.261,148.807
C03014=1234.521,-24.331,-39.455,-179.654,5.261,148.806
C03015=1234.516,-24.082,-39.469,-179.652,5.261,148.805
C03016=1234.511,-23.833,-39.483,-179.649,5.262,148.805
C03017=1234.506,-23.583,-39.496,-179.647,5.261,148.804
C03018=1234.501,-23.333,-39.510,-179.644,5.262,148.803
C03019=1234.496,-23.084,-39.523,-179.642,5.262,148.803
C03020=1234.491,-22.834,-39.537,-179.640,5.262,148.802
C03021=1234.485,-22.565,-39.552,-179.637,5.262,148.801
C03022=1234.480,-22.296,-39.566,-179.634,5.263,148.800
C03023=1234.474,-22.027,-39.581,-179.631,5.263,148.800
C03024=1234.469,-21.757,-39.596,-179.629,5.263,148.799
C03025=1234.464,-21.507,-39.610,-179.626,5.263,148.798
C03026=1234.459,-21.258,-39.623,-179.624,5.264,148.798
C03027=1234.454,-21.008,-39.637,-179.622,5.264,148.797
C03028=1234.448,-20.759,-39.651,-179.619,5.264,148.796
C03029=1234.444,-20.510,-39.664,-179.616,5.264,148.795
C03030=1234.439,-20.259,-39.678,-179.614,5.264,148.795
C03031=1234.433,-20.010,-39.692,-179.611,5.264,148.794
C03032=1234.428,-19.761,-39.706,-179.609,5.264,148.793
C03033=1234.424,-19.510,-39.719,-179.606,5.265,148.792
C03034=1234.418,-19.261,-39.733,-179.604,5.265,148.792
C03035=1234.413,-19.012,-39.747,-179.602,5.265,148.791
C03036=1234.408,-18.762,-39.762,-179.599,5.265,148.790
C03037=1234.403,-18.513,-39.774,-179.596,5.266,148.790
C03038=1234.398,-18.263,-39.789,-179.594,5.266,148.789
C03039=1234.393,-18.013,-39.803,-179.592,5.266,148.788
C03040=1234.387,-17.764,-39.816,-179.589,5.267,148.788
C03041=1234.383,-17.514,-39.830,-179.587,5.266,148.787
C03042=1234.378,-17.265,-39.844,-179.584,5.267,148.786
C03043=1234.372,-17.016,-39.858,-179.582,5.267,148.786
C03044=1234.368,-16.766,-39.872,-179.579,5.267,148.785
C03045=1234.362,-16.516,-39.886,-179.577,5.268,148.784
C03046=1234.357,-16.267,-39.899,-179.575,5.267,148.783
C03047=1234.352,-16.017,-39.913,-179.572,5.268,148.783
C03048=1234.348,-15.767,-39.928,-179.569,5.268,148.782
C03049=1234.342,-15.518,-39.941,-179.567,5.268,148.781
C03050=1234.337,-15.268,-39.955,-179.564,5.268,148.780
C03051=1234.332,-15.019,-39.969,-179.561,5.269,148.780
C03052=1234.328,-14.769,-39.983,-179.559,5.268,148.779
C03053=1234.322,-14.520,-39.997,-179.557,5.269,148.778
C03054=1234.317,-14.270,-40.011,-179.554,5.269,148.778
C03055=1234.312,-14.021,-40.026,-179.552,5.269,148.777
C03056=1234.306,-13.771,-40.039,-179.549,5.270,148.776
C03057=1234.302,-13.522,-40.052,-179.547,5.270,148.776
C03058=1234.297,-13.272,-40.067,-179.545,5.270,148.775
C03059=1234.292,-13.022,-40.081,-179.542,5.270,148.774
C03060=1234.287,-12.773,-40.095,-179.539,5.271,148.773
C03061=1234.282,-12.523,-40.109,-179.537,5.271,148.773
C03062=1234.277,-12.274,-40.123,-179.535,5.271,148.772
C03063=1234.272,-12.024,-40.138,-179.532,5.272,148.771
C03064=1234.266,-11.775,-40.152,-179.530,5.271,148.771
C03065=1234.262,-11.525,-40.165,-179.527,5.272,148.770
C03066=1234.257,-11.275,-40.179,-179.525,5.272,148.769
C03067=1234.252,-11.025,-40.193,-179.522,5.272,148.768
C03068=1234.246,-10.776,-40.207,-179.519,5.272,148.768
C03069=1234.241,-10.527,-40.221,-179.517,5.273,148.767
C03070=1234.236,-10.277,-40.236,-179.515,5.273,148.766
C03071=1234.231,-10.027,-40.250,-179.512,5.273,148.766
C03072=1234.226,-9.778,-40.264,-179.509,5.274,148.765
C03073=1234.221,-9.529,-40.278,-179.507,5.273,148.764
C03074=1234.216,-9.279,-40.292,-179.504,5.274,148.764
C03075=1234.211,-9.029,-40.307,-179.502,5.274,148.763
C03076=1234.206,-8.779,-40.321,-179.500,5.274,148.762
C03077=1234.201,-8.530,-40.335,-179.497,5.275,148.761
C03078=1234.195,-8.281,-40.349,-179.494,5.275,148.761
C03079=1234.190,-8.031,-40.363,-179.492,5.275,148.760
C03080=1234.185,-7.781,-40.378,-179.490,5.275,148.759
C03081=1234.181,-7.532,-40.391,-179.487,5.276,148.759
C03082=1234.177,-7.283,-40.406,-179.485,5.276,148.758
C03083=1234.171,-7.034,-40.420,-179.482,5.276,148.757
C03084=1234.166,-6.784,-40.434,-179.480,5.277,148.757
C03085=1234.161,-6.534,-40.449,-179.478,5.276,148.756
C03086=1234.156,-6.285,-40.463,-179.475,5.277,148.755
C03087=1234.151,-6.035,-40.477,-179.472,5.277,148.755
C03088=1234.146,-5.785,-40.492,-179.470,5.277,148.754
C03089=1234.141,-5.536,-40.506,-179.467,5.277,148.753
C03090=1234.135,-5.286,-40.520,-179.464,5.278,148.752
C03091=1234.130,-5.037,-40.535,-179.462,5.277,148.752
C03092=1234.125,-4.787,-40.550,-179.460,5.278,148.751
C03093=1234.120,-4.538,-40.564,-179.457,5.279,148.750
C03094=1234.115,-4.288,-40.578,-179.455,5.278,148.749
C03095=1234.111,-4.038,-40.592,-179.452,5.279,148.749
C03096=1234.105,-3.789,-40.606,-179.450,5.279,148.748
C03097=1234.100,-3.540,-40.621,-179.448,5.279,148.747
C03098=1234.095,-3.291,-40.636,-179.445,5.280,148.747
C03099=1234.090,-3.041,-40.650,-179.442,5.280,148.746
C03100=1234.085,-2.791,-40.664,-179.440,5.281,148.745
C03101=1234.081,-2.541,-40.678,-179.438,5.280,148.745
C03102=1234.076,-2.292,-40.693,-179.435,5.281,148.744
C03103=1234.071,-2.043,-40.708,-179.432,5.281,148.743
C03104=1234.065,-1.793,-40.723,-179.430,5.281,148.743
C03105=1234.060,-1.544,-40.737,-179.427,5.282,148.742
C03106=1234.055,-1.294,-40.751,-179.425,5.282,148.741
C03107=1234.050,-1.045,-40.766,-179.423,5.282,148.741
C03108=1234.045,-0.795,-40.780,-179.420,5.282,148.740
C03109=1234.040,-0.545,-40.794,-179.417,5.283,148.739
C03110=1234.035,-0.296,-40.809,-179.415,5.283,148.738
C03111=1234.031,-0.047,-40.824,-179.413,5.283,148.738
C03112=1234.025,0.203,-40.839,-179.410,5.284,148.737
C03113=1234.020,0.453,-40.853,-179.407,5.284,148.736
C03114=1234.015,0.703,-40.867,-179.405,5.284,148.736
C03115=1234.010,0.952,-40.882,-179.403,5.284,148.735
C03116=1234.005,1.202,-40.896,-179.400,5.285,148.734
C03117=1234.000,1.451,-40.911,-179.397,5.284,148.733
C03118=1233.994,1.700,-40.926,-179.395,5.285,148.733
C03119=1233.989,1.950,-40.940,-179.392,5.285,148.732
C03120=1233.984,2.200,-40.954,-179.390,5.285,148.731
C03121=1233.980,2.449,-40.969,-179.387,5.286,148.731
C03122=1233.975,2.698,-40.984,-179.385,5.286,148.730
C03123=1233.969,2.948,-40.999,-179.382,5.287,148.729
C03124=1233.965,3.197,-41.014,-179.380,5.286,148.729
C03125=1233.959,3.466,-41.029,-179.377,5.287,148.728
C03126=1233.954,3.735,-41.045,-179.375,5.288,148.727
C03127=1233.948,4.004,-41.061,-179.372,5.288,148.726
C03128=1233.943,4.273,-41.077,-179.369,5.288,148.726
C03129=1233.938,4.523,-41.091,-179.367,5.288,148.725
C03130=1233.933,4.772,-41.107,-179.364,5.289,148.724
C03131=1233.928,5.022,-41.121,-179.362,5.289,148.724
C03132=1233.923,5.271,-41.135,-179.359,5.290,148.723
C03133=1233.918,5.521,-41.150,-179.357,5.289,148.722
C03134=1233.913,5.771,-41.165,-179.354,5.290,148.721
C03135=1233.908,6.020,-41.180,-179.351,5.290,148.721
C03136=1233.903,6.269,-41.195,-179.349,5.290,148.720
C03137=1233.898,6.518,-41.209,-179.347,5.291,148.719
C03138=1233.893,6.768,-41.224,-179.344,5.291,148.719
C03139=1233.888,7.018,-41.239,-179.341,5.292,148.718
C03140=1233.883,7.267,-41.254,-179.339,5.291,148.717
C03141=1233.878,7.517,-41.269,-179.337,5.292,148.717
C03142=1233.873,7.766,-41.284,-179.334,5.293,148.716
C03143=1233.868,8.015,-41.298,-179.331,5.293,148.715
C03144=1233.862,8.266,-41.313,-179.329,5.293,148.715
C03145=1233.858,8.515,-41.328,-179.327,5.293,148.714
C03146=1233.853,8.764,-41.343,-179.324,5.294,148.713
C03147=1233.847,9.014,-41.358,-179.322,5.294,148.713
C03148=1233.843,9.263,-41.373,-179.319,5.294,148.712
C03149=1233.838,9.513,-41.387,-179.317,5.295,148.711
C03150=1233.833,9.763,-41.403,-179.314,5.295,148.710
C03151=1233.828,10.012,-41.418,-179.312,5.295,148.710
C03152=1233.823,10.261,-41.433,-179.309,5.295,148.709
C03153=1233.818,10.511,-41.448,-179.307,5.296,148.708
C03154=1233.813,10.761,-41.463,-179.304,5.297,148.708
C03155=1233.808,11.010,-41.478,-179.302,5.296,148.707
C03156=1233.803,11.259,-41.493,-179.299,5.297,148.706
C03157=1233.798,11.509,-41.507,-179.297,5.297,148.706
C03158=1233.793,11.758,-41.523,-179.294,5.298,148.705
C03159=1233.788,12.008,-41.537,-179.292,5.298,148.704
C03160=1233.782,12.257,-41.553,-179.289,5.298,148.704
C03161=1233.778,12.506,-41.568,-179.287,5.299,148.703
C03162=1233.773,12.757,-41.583,-179.285,5.298,148.702
C03163=1233.768,13.006,-41.598,-179.282,5.299,148.702
C03164=1233.763,13.255,-41.613,-179.279,5.300,148.701
C03165=1233.758,13.505,-41.629,-179.277,5.300,148.700
C03166=1233.753,13.754,-41.643,-179.275,5.300,148.700
C03167=1233.748,14.004,-41.659,-179.272,5.300,148.699
C03168=1233.743,14.253,-41.674,-179.269,5.301,148.698
C03169=1233.737,14.503,-41.688,-179.267,5.301,148.697
C03170=1233.733,14.753,-41.704,-179.264,5.301,148.697
C03171=1233.729,15.002,-41.719,-179.262,5.302,148.696
C03172=1233.723,15.251,-41.734,-179.259,5.302,148.695
C03173=1233.718,15.501,-41.749,-179.257,5.303,148.695
C03174=1233.713,15.750,-41.764,-179.254,5.303,148.694
C03175=1233.708,15.999,-41.779,-179.252,5.303,148.693
C03176=1233.703,16.249,-41.795,-179.249,5.304,148.693
C03177=1233.699,16.499,-41.810,-179.247,5.304,148.692
C03178=1233.693,16.749,-41.825,-179.244,5.305,148.691
C03179=1233.688,16.998,-41.840,-179.241,5.304,148.690
C03180=1233.683,17.247,-41.856,-179.239,5.305,148.690
C03181=1233.678,17.496,-41.871,-179.236,5.305,148.689
C03182=1233.673,17.746,-41.886,-179.233,5.306,148.688
C03183=1233.668,17.996,-41.902,-179.231,5.305,148.688
C03184=1233.663,18.245,-41.916,-179.229,5.306,148.687
C03185=1233.658,18.495,-41.932,-179.226,5.307,148.687
C03186=1233.653,18.744,-41.947,-179.224,5.307,148.686
C03187=1233.648,18.993,-41.963,-179.222,5.307,148.685
C03188=1233.644,19.243,-41.978,-179.219,5.308,148.684
C03189=1233.638,19.492,-41.994,-179.216,5.308,148.684
C03190=1233.633,19.742,-42.009,-179.214,5.309,148.683
C03191=1233.628,19.991,-42.024,-179.212,5.309,148.682
C03192=1233.623,20.241,-42.039,-179.209,5.309,148.682
C03193=1233.619,20.491,-42.054,-179.206,5.310,148.681
C03194=1233.613,20.740,-42.070,-179.204,5.310,148.680
C03195=1233.608,20.990,-42.086,-179.201,5.311,148.680
C03196=1233.603,21.239,-42.101,-179.199,5.310,148.679
C03197=1233.598,21.489,-42.116,-179.196,5.311,148.678
C03198=1233.594,21.738,-42.131,-179.194,5.312,148.678
C03199=1233.588,21.987,-42.147,-179.191,5.312,148.677
C03200=1233.583,22.237,-42.163,-179.189,5.312,148.676
C03201=1233.578,22.486,-42.178,-179.186,5.312,148.676
C03202=1233.574,22.736,-42.194,-179.184,5.313,148.675
C03203=1233.568,22.985,-42.209,-179.181,5.314,148.674
C03204=1233.564,23.234,-42.224,-179.178,5.314,148.674
C03205=1233.558,23.484,-42.240,-179.176,5.314,148.673
C03206=1233.553,23.734,-42.256,-179.174,5.314,148.672
C03207=1233.549,23.983,-42.271,-179.171,5.315,148.672
C03208=1233.543,24.232,-42.286,-179.168,5.315,148.671
C03209=1233.539,24.482,-42.302,-179.166,5.315,148.670
C03210=1233.534,24.732,-42.317,-179.164,5.316,148.669
C03211=1233.529,24.981,-42.333,-179.161,5.316,148.669
C03212=1233.523,25.230,-42.348,-179.158,5.317,148.668
C03213=1233.519,25.480,-42.365,-179.156,5.317,148.667
C03214=1233.514,25.729,-42.380,-179.154,5.317,148.667
C03215=1233.509,25.978,-42.396,-179.151,5.318,148.666
C03216=1233.504,26.228,-42.412,-179.148,5.318,148.665
C03217=1233.499,26.478,-42.427,-179.146,5.319,148.665
C03218=1233.494,26.727,-42.442,-179.143,5.319,148.664
C03219=1233.489,26.977,-42.458,-179.141,5.319,148.663
C03220=1233.484,27.226,-42.474,-179.138,5.320,148.663
C03221=1233.479,27.476,-42.489,-179.136,5.320,148.662
C03222=1233.474,27.724,-42.505,-179.133,5.321,148.661
C03223=1233.469,27.974,-42.521,-179.131,5.321,148.661
C03224=1233.464,28.224,-42.537,-179.128,5.321,148.660
C03225=1233.459,28.473,-42.552,-179.126,5.322,148.659
C03226=1233.454,28.723,-42.568,-179.123,5.322,148.659
C03227=1233.449,28.972,-42.583,-179.121,5.323,148.658
C03228=1233.444,29.221,-42.599,-179.118,5.323,148.657
C03229=1233.439,29.490,-42.617,-179.115,5.324,148.657
C03230=1233.434,29.759,-42.633,-179.113,5.324,148.656
C03231=1233.429,30.027,-42.650,-179.111,5.324,148.655
C03232=1233.423,30.296,-42.667,-179.107,5.324,148.654
C03233=1233.418,30.546,-42.683,-179.105,5.325,148.654
C03234=1233.413,30.795,-42.699,-179.102,5.325,148.653
C03235=1233.407,31.044,-42.714,-179.099,5.326,148.652
C03236=1233.404,31.294,-42.730,-179.097,5.327,148.652
C03237=1233.398,31.543,-42.746,-179.095,5.327,148.651
C03238=1233.393,31.793,-42.762,-179.093,5.327,148.650
C03239=1233.388,32.043,-42.778,-179.090,5.328,148.650
C03240=1233.383,32.291,-42.794,-179.087,5.328,148.649
C03241=1233.378,32.541,-42.810,-179.085,5.329,148.648
C03242=1233.373,32.791,-42.825,-179.082,5.329,148.648
C03243=1233.368,33.039,-42.841,-179.080,5.329,148.647
C03244=1233.364,33.289,-42.857,-179.077,5.330,148.646
C03245=1233.358,33.539,-42.873,-179.075,5.330,148.646
C03246=1233.354,33.788,-42.889,-179.072,5.331,148.645
C03247=1233.348,34.038,-42.905,-179.069,5.331,148.644
C03248=1233.344,34.288,-42.921,-179.067,5.332,148.644
C03249=1233.339,34.537,-42.937,-179.065,5.332,148.643
C03250=1233.333,34.786,-42.953,-179.062,5.332,148.642
C03251=1233.328,35.036,-42.969,-179.059,5.333,148.642
C03252=1233.323,35.285,-42.985,-179.057,5.333,148.641
C03253=1233.319,35.535,-43.001,-179.054,5.334,148.640
C03254=1233.313,35.784,-43.017,-179.051,5.335,148.640
C03255=1233.309,36.034,-43.033,-179.049,5.334,148.639
C03256=1233.304,36.282,-43.049,-179.047,5.335,148.638
C03257=1233.299,36.532,-43.065,-179.044,5.335,148.638
C03258=1233.294,36.782,-43.081,-179.041,5.336,148.637
C03259=1233.289,37.031,-43.097,-179.039,5.337,148.636
C03260=1233.284,37.281,-43.113,-179.037,5.337,148.636
C03261=1233.279,37.529,-43.129,-179.035,5.337,148.635
C03262=1233.274,37.780,-43.145,-179.032,5.338,148.634
C03263=1233.269,38.028,-43.161,-179.029,5.338,148.634
C03264=1233.265,38.278,-43.177,-179.027,5.339,148.633
C03265=1233.259,38.527,-43.194,-179.024,5.339,148.632
C03266=1233.255,38.777,-43.210,-179.021,5.340,148.632
C03267=1233.250,39.026,-43.226,-179.019,5.340,148.631
C03268=1233.245,39.276,-43.242,-179.017,5.340,148.630
C03269=1233.240,39.525,-43.258,-179.014,5.341,148.630
C03270=1233.235,39.775,-43.274,-179.011,5.341,148.629
C03271=1233.230,40.024,-43.290,-179.009,5.342,148.628
C03272=1233.225,40.274,-43.306,-179.006,5.343,148.628
C03273=1233.219,40.523,-43.323,-179.003,5.343,148.627
C03274=1233.215,40.773,-43.340,-179.001,5.343,148.626
C03275=1233.209,41.022,-43.355,-178.999,5.343,148.626
C03276=1233.205,41.271,-43.372,-178.996,5.344,148.625
C03277=1233.200,41.521,-43.388,-178.993,5.345,148.624
C03278=1233.195,41.770,-43.404,-178.991,5.346,148.624
C03279=1233.190,42.019,-43.421,-178.989,5.346,148.623
C03280=1233.185,42.269,-43.437,-178.986,5.347,148.623
C03281=1233.180,42.518,-43.453,-178.984,5.346,148.622
C03282=1233.175,42.768,-43.469,-178.981,5.347,148.621
C03283=1233.170,43.017,-43.485,-178.979,5.348,148.620
C03284=1233.166,43.266,-43.502,-178.976,5.348,148.620
C03285=1233.160,43.517,-43.518,-178.973,5.349,148.619
C03286=1233.155,43.766,-43.535,-178.971,5.349,148.618
C03287=1233.151,44.015,-43.551,-178.968,5.350,148.618
C03288=1233.145,44.264,-43.567,-178.966,5.350,148.617
C03289=1233.141,44.514,-43.584,-178.963,5.350,148.616
C03290=1233.136,44.763,-43.600,-178.961,5.351,148.616
C03291=1233.131,45.012,-43.617,-178.958,5.351,148.615
C03292=1233.125,45.262,-43.633,-178.956,5.352,148.615
C03293=1233.121,45.511,-43.649,-178.953,5.353,148.614
C03294=1233.116,45.761,-43.666,-178.951,5.353,148.613
C03295=1233.111,46.010,-43.682,-178.948,5.354,148.613
C03296=1233.106,46.260,-43.698,-178.946,5.354,148.612
C03297=1233.101,46.509,-43.715,-178.943,5.354,148.611
C03298=1233.096,46.758,-43.732,-178.941,5.355,148.611
C03299=1233.092,47.008,-43.749,-178.938,5.355,148.610
C03300=1233.086,47.257,-43.764,-178.935,5.356,148.609
C03301=1233.082,47.507,-43.781,-178.933,5.357,148.609
C03302=1233.077,47.756,-43.798,-178.930,5.357,148.608
C03303=1233.071,48.005,-43.814,-178.928,5.358,148.607
C03304=1233.067,48.255,-43.831,-178.925,5.359,148.607
C03305=1233.061,48.504,-43.847,-178.923,5.358,148.606
C03306=1233.057,48.754,-43.863,-178.921,5.359,148.605
C03307=1233.052,49.004,-43.881,-178.918,5.360,148.605
C03308=1233.047,49.252,-43.897,-178.915,5.360,148.604
C03309=1233.042,49.502,-43.914,-178.913,5.361,148.603
C03310=1233.038,49.751,-43.930,-178.910,5.361,148.603
C03311=1233.032,50.000,-43.947,-178.908,5.362,148.602
C03312=1233.027,50.250,-43.963,-178.905,5.362,148.601
C03313=1233.023,50.500,-43.980,-178.902,5.363,148.601
C03314=1233.018,50.749,-43.996,-178.900,5.363,148.600
C03315=1233.012,50.999,-44.013,-178.898,5.363,148.599
C03316=1233.008,51.248,-44.030,-178.895,5.364,148.599
C03317=1233.003,51.497,-44.046,-178.893,5.365,148.598
C03318=1232.998,51.747,-44.064,-178.890,5.365,148.598
C03319=1232.993,51.996,-44.080,-178.888,5.366,148.597
C03320=1232.988,52.245,-44.097,-178.885,5.367,148.596
C03321=1232.983,52.495,-44.114,-178.882,5.367,148.596
C03322=1232.978,52.744,-44.131,-178.880,5.368,148.595
C03323=1232.973,52.993,-44.147,-178.877,5.368,148.594
C03324=1232.968,53.243,-44.164,-178.875,5.368,148.594
C03325=1232.964,53.492,-44.181,-178.872,5.369,148.593
C03326=1232.959,53.742,-44.197,-178.870,5.370,148.593
C03327=1232.953,53.991,-44.214,-178.867,5.370,148.592
C03328=1232.949,54.240,-44.231,-178.865,5.371,148.591
C03329=1232.944,54.490,-44.248,-178.862,5.371,148.591
C03330=1232.938,54.739,-44.265,-178.860,5.372,148.590
C03331=1232.934,54.988,-44.281,-178.857,5.372,148.589
C03332=1232.930,55.238,-44.298,-178.854,5.373,148.589
C03333=1232.924,55.506,-44.316,-178.852,5.374,148.588
C03334=1232.919,55.775,-44.334,-178.849,5.374,148.587
C03335=1232.913,56.043,-44.353,-178.846,5.375,148.587
C03336=1232.908,56.311,-44.371,-178.844,5.375,148.586
C03337=1232.903,56.561,-44.388,-178.841,5.376,148.585
C03338=1232.898,56.810,-44.404,-178.839,5.376,148.585
C03339=1232.893,57.060,-44.422,-178.836,5.377,148.584
C03340=1232.888,57.309,-44.438,-178.833,5.378,148.583
C03341=1232.884,57.559,-44.455,-178.831,5.378,148.583
C03342=1232.879,57.808,-44.472,-178.828,5.379,148.582
C03343=1232.873,58.057,-44.489,-178.826,5.379,148.581
C03344=1232.869,58.306,-44.506,-178.824,5.379,148.581
C03345=1232.864,58.556,-44.523,-178.821,5.380,148.580
C03346=1232.859,58.806,-44.540,-178.818,5.381,148.579
C03347=1232.854,59.054,-44.557,-178.816,5.381,148.579
C03348=1232.849,59.304,-44.574,-178.813,5.382,148.578
C03349=1232.844,59.554,-44.591,-178.811,5.382,148.577
C03350=1232.839,59.803,-44.609,-178.808,5.383,148.577
C03351=1232.835,60.052,-44.625,-178.806,5.384,148.576
C03352=1232.829,60.301,-44.642,-178.803,5.385,148.576
C03353=1232.824,60.551,-44.659,-178.801,5.385,148.575
C03354=1232.819,60.801,-44.676,-178.798,5.386,148.574
C03355=1232.815,61.050,-44.694,-178.795,5.386,148.574
C03356=1232.810,61.299,-44.711,-178.793,5.387,148.573
C03357=1232.805,61.548,-44.727,-178.790,5.387,148.572
C03358=1232.800,61.797,-44.745,-178.787,5.388,148.572
C03359=1232.795,62.047,-44.762,-178.785,5.389,148.571
C03360=1232.790,62.297,-44.779,-178.783,5.389,148.571
C03361=1232.785,62.546,-44.796,-178.781,5.389,148.570
C03362=1232.781,62.795,-44.814,-178.778,5.390,148.569
C03363=1232.775,63.044,-44.831,-178.775,5.390,148.569
C03364=1232.770,63.294,-44.847,-178.773,5.391,148.568
C03365=1232.765,63.543,-44.865,-178.770,5.392,148.567
C03366=1232.761,63.793,-44.882,-178.768,5.393,148.567
C03367=1232.756,64.042,-44.899,-178.765,5.393,148.566
C03368=1232.751,64.291,-44.917,-178.763,5.394,148.565
C03369=1232.746,64.541,-44.934,-178.760,5.394,148.565
C03370=1232.741,64.791,-44.951,-178.757,5.395,148.564
C03371=1232.736,65.039,-44.968,-178.755,5.396,148.563
C03372=1232.731,65.289,-44.985,-178.752,5.396,148.563
C03373=1232.726,65.538,-45.003,-178.750,5.397,148.562
C03374=1232.722,65.787,-45.020,-178.747,5.398,148.562
C03375=1232.717,66.037,-45.037,-178.745,5.398,148.561
C03376=1232.712,66.286,-45.055,-178.742,5.399,148.560
C03377=1232.707,66.536,-45.072,-178.739,5.399,148.560
C03378=1232.702,66.785,-45.090,-178.737,5.400,148.559
C03379=1232.697,67.035,-45.107,-178.734,5.401,148.558
C03380=1232.692,67.283,-45.124,-178.732,5.402,148.558
C03381=1232.687,67.533,-45.141,-178.729,5.402,148.557
C03382=1232.682,67.783,-45.159,-178.727,5.403,148.557
C03383=1232.678,68.031,-45.176,-178.724,5.403,148.556
C03384=1232.672,68.281,-45.193,-178.722,5.404,148.555
C03385=1232.668,68.530,-45.211,-178.719,5.404,148.555
C03386=1232.663,68.780,-45.228,-178.717,5.405,148.554
C03387=1232.658,69.029,-45.246,-178.715,5.405,148.554
C03388=1232.653,69.278,-45.264,-178.712,5.406,148.553
C03389=1232.649,69.528,-45.281,-178.709,5.406,148.552
C03390=1232.644,69.777,-45.299,-178.707,5.407,148.552
C03391=1232.639,70.027,-45.316,-178.704,5.408,148.551
C03392=1232.634,70.276,-45.334,-178.702,5.408,148.550
C03393=1232.629,70.525,-45.351,-178.699,5.409,148.550
C03394=1232.624,70.775,-45.368,-178.697,5.410,148.549
C03395=1232.619,71.024,-45.386,-178.694,5.410,148.548
C03396=1232.614,71.274,-45.404,-178.692,5.411,148.548
C03397=1232.610,71.522,-45.421,-178.689,5.411,148.547
C03398=1232.605,71.772,-45.438,-178.687,5.412,148.547
C03399=1232.600,72.021,-45.456,-178.684,5.413,148.546
C03400=1232.595,72.271,-45.474,-178.682,5.414,148.545
C03401=1232.590,72.520,-45.492,-178.679,5.414,148.545
C03402=1232.586,72.769,-45.509,-178.676,5.415,148.544
C03403=1232.580,73.019,-45.526,-178.674,5.415,148.543
C03404=1232.575,73.268,-45.544,-178.671,5.416,148.543
C03405=1232.571,73.517,-45.562,-178.669,5.417,148.542
C03406=1232.565,73.767,-45.579,-178.666,5.417,148.542
C03407=1232.561,74.016,-45.597,-178.664,5.418,148.541
C03408=1232.556,74.265,-45.615,-178.661,5.419,148.540
C03409=1232.551,74.515,-45.632,-178.659,5.420,148.540
C03410=1232.546,74.764,-45.650,-178.656,5.420,148.539
C03411=1232.541,75.013,-45.668,-178.654,5.421,148.539
C03412=1232.536,75.262,-45.686,-178.651,5.421,148.538
C03413=1232.531,75.512,-45.703,-178.648,5.422,148.537
C03414=1232.527,75.761,-45.721,-178.646,5.423,148.537
C03415=1232.522,76.010,-45.739,-178.644,5.424,148.536
C03416=1232.517,76.259,-45.757,-178.641,5.424,148.536
C03417=1232.512,76.509,-45.774,-178.638,5.425,148.535
C03418=1232.507,76.758,-45.792,-178.636,5.425,148.534
C03419=1232.502,77.008,-45.810,-178.633,5.426,148.534
C03420=1232.497,77.257,-45.828,-178.631,5.427,148.533
C03421=1232.492,77.507,-45.845,-178.628,5.428,148.533
C03422=1232.487,77.756,-45.863,-178.625,5.429,148.532
C03423=1232.482,78.005,-45.881,-178.622,5.429,148.531
C03424=1232.478,78.254,-45.898,-178.620,5.430,148.531
C03425=1232.473,78.503,-45.916,-178.618,5.431,148.530
C03426=1232.469,78.753,-45.935,-178.615,5.432,148.529
C03427=1232.463,79.003,-45.952,-178.612,5.432,148.529
C03428=1232.459,79.252,-45.970,-178.610,5.433,148.528
C03429=1232.454,79.501,-45.988,-178.607,5.433,148.527
C03430=1232.449,79.750,-46.006,-178.605,5.434,148.527
C03431=1232.444,79.999,-46.024,-178.602,5.435,148.526
C03432=1232.439,80.249,-46.042,-178.600,5.436,148.526
C03433=1232.434,80.498,-46.060,-178.597,5.436,148.525
C03434=1232.429,80.747,-46.078,-178.595,5.437,148.524
C03435=1232.424,80.996,-46.096,-178.592,5.438,148.524
C03436=1232.420,81.246,-46.114,-178.590,5.438,148.523
C03437=1232.414,81.515,-46.133,-178.587,5.439,148.523
C03438=1232.409,81.783,-46.152,-178.585,5.440,148.522
C03439=1232.404,82.051,-46.172,-178.581,5.441,148.521
C03440=1232.398,82.320,-46.192,-178.579,5.442,148.521
C03441=1232.394,82.569,-46.210,-178.576,5.442,148.520
C03442=1232.389,82.818,-46.228,-178.574,5.443,148.519
C03443=1232.384,83.067,-46.246,-178.571,5.443,148.519
C03444=1232.379,83.317,-46.264,-178.569,5.444,148.518
C03445=1232.374,83.566,-46.282,-178.566,5.445,148.518
C03446=1232.370,83.816,-46.300,-178.564,5.446,148.517
C03447=1232.365,84.065,-46.318,-178.561,5.446,148.516
C03448=1232.360,84.314,-46.336,-178.559,5.447,148.516
C03449=1232.355,84.563,-46.354,-178.556,5.448,148.515
C03450=1232.350,84.812,-46.372,-178.554,5.448,148.515
C03451=1232.345,85.062,-46.390,-178.551,5.449,148.514
C03452=1232.341,85.311,-46.408,-178.549,5.450,148.514
C03453=1232.335,85.561,-46.427,-178.546,5.450,148.513
C03454=1232.330,85.810,-46.445,-178.543,5.452,148.512
C03455=1232.326,86.059,-46.464,-178.540,5.452,148.512
C03456=1232.321,86.308,-46.481,-178.538,5.453,148.511
C03457=1232.316,86.558,-46.500,-178.536,5.454,148.511
C03458=1232.311,86.807,-46.518,-178.533,5.455,148.510
C03459=1232.307,87.056,-46.536,-178.530,5.455,148.509
C03460=1232.302,87.305,-46.554,-178.528,5.456,148.509
C03461=1232.296,87.555,-46.572,-178.526,5.457,148.508
C03462=1232.292,87.805,-46.591,-178.523,5.457,148.507
C03463=1232.287,88.053,-46.609,-178.520,5.458,148.507
C03464=1232.282,88.302,-46.627,-178.518,5.459,148.506
C03465=1232.277,88.551,-46.645,-178.516,5.460,148.506
C03466=1232.273,88.801,-46.664,-178.513,5.460,148.505
C03467=1232.267,89.051,-46.682,-178.510,5.461,148.504
C03468=1232.263,89.299,-46.701,-178.508,5.461,148.504
C03469=1232.258,89.549,-46.719,-178.505,5.463,148.503
C03470=1232.253,89.798,-46.737,-178.502,5.464,148.503
C03471=1232.249,90.048,-46.755,-178.500,5.464,148.502
C03472=1232.243,90.296,-46.775,-178.497,5.465,148.501
C03473=1232.238,90.546,-46.793,-178.495,5.466,148.501
C03474=1232.234,90.796,-46.811,-178.492,5.467,148.500
C03475=1232.229,91.045,-46.829,-178.490,5.467,148.500
C03476=1232.224,91.294,-46.848,-178.487,5.468,148.499
C03477=1232.219,91.543,-46.866,-178.485,5.469,148.499
C03478=1232.214,91.793,-46.884,-178.482,5.469,148.498
C03479=1232.210,92.041,-46.903,-178.480,5.470,148.497
C03480=1232.204,92.291,-46.922,-178.477,5.471,148.497
C03481=1232.200,92.541,-46.940,-178.474,5.472,148.496
C03482=1232.195,92.789,-46.959,-178.472,5.473,148.496
C03483=1232.190,93.038,-46.977,-178.469,5.474,148.495
C03484=1232.185,93.288,-46.996,-178.467,5.474,148.494
C03485=1232.181,93.537,-47.014,-178.465,5.475,148.494
C03486=1232.176,93.786,-47.032,-178.462,5.476,148.493
C03487=1232.171,94.036,-47.051,-178.459,5.476,148.493
C03488=1232.166,94.285,-47.070,-178.457,5.477,148.492
C03489=1232.161,94.534,-47.088,-178.455,5.478,148.492
C03490=1232.156,94.784,-47.108,-178.451,5.479,148.491
C03491=1232.152,95.033,-47.126,-178.449,5.480,148.490
C03492=1232.147,95.282,-47.144,-178.447,5.481,148.490
C03493=1232.142,95.532,-47.163,-178.444,5.482,148.489
C03494=1232.137,95.781,-47.181,-178.441,5.482,148.489
C03495=1232.132,96.029,-47.200,-178.439,5.483,148.488
C03496=1232.127,96.280,-47.219,-178.437,5.484,148.487
C03497=1232.123,96.528,-47.238,-178.434,5.484,148.487
C03498=1232.118,96.777,-47.256,-178.431,5.485,148.486
C03499=1232.113,97.027,-47.275,-178.429,5.487,148.486
C03500=1232.108,97.276,-47.293,-178.426,5.487,148.485
C03501=1232.103,97.525,-47.312,-178.423,5.488,148.484
C03502=1232.099,97.775,-47.331,-178.421,5.489,148.484
C03503=1232.094,98.023,-47.350,-178.419,5.490,148.483
C03504=1232.089,98.274,-47.368,-178.416,5.490,148.483
C03505=1232.084,98.522,-47.387,-178.413,5.491,148.482
C03506=1232.079,98.772,-47.406,-178.411,5.492,148.482
C03507=1232.075,99.021,-47.425,-178.408,5.493,148.481
C03508=1232.069,99.270,-47.443,-178.406,5.494,148.480
C03509=1232.065,99.520,-47.462,-178.403,5.494,148.480
C03510=1232.060,99.769,-47.480,-178.401,5.495,148.479
C03511=1232.055,100.018,-47.500,-178.398,5.496,148.479
C03512=1232.051,100.267,-47.519,-178.396,5.497,148.478
C03513=1232.045,100.516,-47.537,-178.393,5.498,148.478
C03514=1232.041,100.766,-47.556,-178.390,5.499,148.477
C03515=1232.035,101.015,-47.575,-178.388,5.500,148.476
C03516=1232.031,101.264,-47.594,-178.385,5.500,148.476
C03517=1232.026,101.513,-47.613,-178.383,5.501,148.475
C03518=1232.021,101.762,-47.631,-178.380,5.502,148.475
C03519=1232.016,102.012,-47.651,-178.378,5.502,148.474
C03520=1232.012,102.260,-47.670,-178.376,5.503,148.474
C03521=1232.007,102.511,-47.689,-178.372,5.505,148.473
C03522=1232.002,102.759,-47.707,-178.370,5.505,148.472
C03523=1231.997,103.009,-47.727,-178.368,5.506,148.472
C03524=1231.993,103.257,-47.746,-178.365,5.507,148.471
C03525=1231.988,103.508,-47.765,-178.362,5.508,148.471
C03526=1231.982,103.756,-47.784,-178.360,5.509,148.470
C03527=1231.978,104.006,-47.803,-178.358,5.509,148.469
C03528=1231.973,104.255,-47.822,-178.354,5.511,148.469
C03529=1231.969,104.504,-47.841,-178.352,5.512,148.468
C03530=1231.963,104.753,-47.860,-178.350,5.512,148.468
C03531=1231.959,105.003,-47.879,-178.347,5.513,148.467
C03532=1231.954,105.252,-47.898,-178.345,5.514,148.466
C03533=1231.949,105.502,-47.917,-178.342,5.514,148.466
C03534=1231.944,105.750,-47.936,-178.339,5.516,148.465
C03535=1231.940,106.000,-47.956,-178.337,5.517,148.465
C03536=1231.935,106.248,-47.974,-178.334,5.517,148.464
C03537=1231.930,106.498,-47.994,-178.332,5.518,148.464
C03538=1231.925,106.747,-48.012,-178.329,5.519,148.463
C03539=1231.921,106.997,-48.032,-178.327,5.520,148.463
C03540=1231.915,107.245,-48.051,-178.324,5.521,148.462
C03541=1231.910,107.514,-48.072,-178.321,5.522,148.461
C03542=1231.905,107.783,-48.092,-178.319,5.522,148.461
C03543=1231.900,108.051,-48.113,-178.316,5.524,148.460
C03544=1231.895,108.319,-48.133,-178.313,5.525,148.460
C03545=1231.890,108.569,-48.153,-178.311,5.525,148.459
C03546=1231.885,108.818,-48.172,-178.308,5.526,148.458
C03547=1231.881,109.067,-48.191,-178.305,5.528,148.458
C03548=1231.876,109.316,-48.211,-178.303,5.528,148.457
C03549=1231.871,109.565,-48.230,-178.300,5.529,148.457
C03550=1231.866,109.815,-48.250,-178.298,5.530,148.456
C03551=1231.861,110.064,-48.268,-178.296,5.531,148.456
C03552=1231.856,110.313,-48.287,-178.293,5.531,148.455
C03553=1231.852,110.563,-48.307,-178.290,5.533,148.455
C03554=1231.847,110.812,-48.326,-178.288,5.534,148.454
C03555=1231.842,111.061,-48.345,-178.285,5.534,148.453
C03556=1231.837,111.310,-48.365,-178.283,5.535,148.453
C03557=1231.832,111.560,-48.384,-178.280,5.536,148.452
C03558=1231.828,111.809,-48.403,-178.277,5.537,148.452
C03559=1231.823,112.058,-48.423,-178.275,5.538,148.451
C03560=1231.818,112.307,-48.442,-178.272,5.539,148.451
C03561=1231.813,112.556,-48.462,-178.270,5.540,148.450
C03562=1231.809,112.805,-48.481,-178.268,5.541,148.450
C03563=1231.804,113.054,-48.501,-178.264,5.542,148.449
C03564=1231.799,113.303,-48.520,-178.262,5.543,148.449
C03565=1231.794,113.553,-48.540,-178.260,5.544,148.448
C03566=1231.789,113.802,-48.559,-178.257,5.544,148.447
C03567=1231.785,114.051,-48.578,-178.255,5.545,148.447
C03568=1231.780,114.300,-48.598,-178.252,5.547,148.446
C03569=1231.775,114.549,-48.617,-178.249,5.547,148.446
C03570=1231.770,114.799,-48.637,-178.247,5.548,148.445
C03571=1231.765,115.048,-48.657,-178.244,5.549,148.445
C03572=1231.761,115.297,-48.675,-178.242,5.551,148.444
C03573=1231.756,115.546,-48.696,-178.239,5.551,148.443
C03574=1231.751,115.796,-48.715,-178.237,5.552,148.443
C03575=1231.746,116.044,-48.735,-178.234,5.553,148.442
C03576=1231.741,116.294,-48.754,-178.232,5.554,148.442
C03577=1231.737,116.544,-48.774,-178.229,5.555,148.441
C03578=1231.732,116.792,-48.794,-178.227,5.556,148.441
C03579=1231.727,117.041,-48.814,-178.224,5.557,148.440
C03580=1231.723,117.291,-48.833,-178.222,5.558,148.440
C03581=1231.717,117.539,-48.852,-178.219,5.559,148.439
C03582=1231.713,117.789,-48.872,-178.216,5.560,148.438
C03583=1231.708,118.038,-48.892,-178.214,5.561,148.438
C03584=1231.704,118.288,-48.912,-178.211,5.561,148.437
C03585=1231.698,118.536,-48.931,-178.209,5.562,148.437
C03586=1231.693,118.786,-48.951,-178.206,5.564,148.436
C03587=1231.689,119.035,-48.971,-178.203,5.564,148.436
C03588=1231.684,119.284,-48.990,-178.201,5.565,148.435
C03589=1231.679,119.533,-49.010,-178.199,5.566,148.435
C03590=1231.675,119.782,-49.030,-178.196,5.567,148.434
C03591=1231.670,120.032,-49.050,-178.193,5.568,148.434
C03592=1231.664,120.281,-49.069,-178.191,5.569,148.433
C03593=1231.660,120.530,-49.090,-178.189,5.570,148.433
C03594=1231.655,120.779,-49.109,-178.186,5.571,148.432
C03595=1231.651,121.029,-49.128,-178.183,5.572,148.431
C03596=1231.646,121.277,-49.148,-178.181,5.573,148.431
C03597=1231.641,121.526,-49.168,-178.178,5.574,148.430
C03598=1231.637,121.776,-49.188,-178.176,5.576,148.430
C03599=1231.632,122.025,-49.208,-178.173,5.576,148.429
C03600=1231.627,122.274,-49.227,-178.170,5.577,148.429
C03601=1231.622,122.523,-49.248,-178.168,5.578,148.428
C03602=1231.617,122.773,-49.268,-178.165,5.579,148.428
C03603=1231.612,123.022,-49.288,-178.163,5.580,148.427
C03604=1231.607,123.270,-49.308,-178.160,5.581,148.427
C03605=1231.602,123.520,-49.327,-178.158,5.581,148.426
C03606=1231.598,123.769,-49.348,-178.155,5.583,148.426
C03607=1231.593,124.018,-49.367,-178.152,5.584,148.425
C03608=1231.589,124.267,-49.388,-178.150,5.585,148.424
C03609=1231.584,124.516,-49.407,-178.147,5.586,148.424
C03610=1231.579,124.765,-49.427,-178.145,5.587,148.423
C03611=1231.574,125.015,-49.447,-178.142,5.588,148.423
C03612=1231.570,125.264,-49.467,-178.140,5.589,148.422
C03613=1231.565,125.513,-49.487,-178.137,5.590,148.422
C03614=1231.561,125.762,-49.507,-178.135,5.591,148.421
C03615=1231.555,126.011,-49.527,-178.132,5.592,148.421
C03616=1231.550,126.260,-49.548,-178.130,5.593,148.420
C03617=1231.545,126.510,-49.567,-178.127,5.594,148.420
C03618=1231.541,126.759,-49.588,-178.125,5.595,148.419
C03619=1231.536,127.008,-49.607,-178.122,5.596,148.418
C03620=1231.532,127.257,-49.628,-178.119,5.598,148.418
C03621=1231.527,127.506,-49.648,-178.117,5.598,148.417
C03622=1231.522,127.755,-49.667,-178.115,5.599,148.417
C03623=1231.518,128.004,-49.688,-178.112,5.600,148.416
C03624=1231.512,128.254,-49.708,-178.109,5.602,148.416
C03625=1231.508,128.503,-49.728,-178.107,5.602,148.415
C03626=1231.503,128.752,-49.749,-178.104,5.603,148.415
C03627=1231.499,129.002,-49.768,-178.101,5.605,148.414
C03628=1231.494,129.250,-49.789,-178.099,5.605,148.414
C03629=1231.489,129.499,-49.809,-178.097,5.606,148.413
C03630=1231.484,129.749,-49.829,-178.094,5.607,148.413
C03631=1231.479,129.998,-49.849,-178.091,5.609,148.412
C03632=1231.475,130.246,-49.870,-178.089,5.609,148.412
C03633=1231.470,130.496,-49.889,-178.087,5.610,148.411
C03634=1231.465,130.745,-49.910,-178.083,5.612,148.411
C03635=1231.460,130.994,-49.931,-178.081,5.613,148.410
C03636=1231.456,131.243,-49.951,-178.079,5.613,148.410
C03637=1231.451,131.493,-49.971,-178.076,5.615,148.409
C03638=1231.446,131.742,-49.992,-178.073,5.616,148.409
C03639=1231.441,131.990,-50.012,-178.071,5.617,148.408
C03640=1231.437,132.239,-50.032,-178.068,5.618,148.408
C03641=1231.432,132.489,-50.052,-178.066,5.619,148.407
C03642=1231.427,132.738,-50.073,-178.064,5.620,148.407
C03643=1231.422,132.987,-50.093,-178.061,5.621,148.406
C03644=1231.418,133.236,-50.113,-178.058,5.622,148.406
C03645=1231.412,133.505,-50.135,-178.056,5.623,148.405
C03646=1231.407,133.774,-50.158,-178.052,5.625,148.404
C03647=1231.402,134.043,-50.179,-178.050,5.625,148.404
C03648=1231.397,134.311,-50.201,-178.047,5.627,148.403
C03649=1231.393,134.560,-50.222,-178.045,5.628,148.403
C03650=1231.387,134.809,-50.243,-178.042,5.629,148.402
